# B&R Automation Studio project TD52 (part 80)

#### LamCtrPBC.h
```c
/********************************************************************
 * COPYRIGHT -- B&R Industrial Automation GmbH
 ********************************************************************
 * Program: LamCtrPBC
 * File: LamCtrPBC.h
 * Author: kafkama00
 * Last modified by: kafkama00
 * Created: Mon Oct 11 17:08:29 2021
 * Last modified: Wed Dec 01 09:46:51 2021
 * Model Version: 1.00
 * Description: Lambda controller for pressure based control engines
 * modified Comment: V0.01 11.10.2021 created for first tests
   V0.02 12.10.2021 added debug signals
   V0.03 17.11.2021 added distortion rejection
   V1.00 01.12.2021 remove distortion rejection, serial release DIA.NE V4.11
 ********************************************************************
 * Header for program LamCtrPBC
 ********************************************************************
 * Generated with B&R Automation Studio Target for Simulink V6.4.1
 * (ERT based)
 ********************************************************************/

#ifndef RTW_HEADER_LamCtrPBC_h_
#define RTW_HEADER_LamCtrPBC_h_
#include <math.h>
#include <string.h>
#ifndef LamCtrPBC_COMMON_INCLUDES_
# define LamCtrPBC_COMMON_INCLUDES_
#include "rtwtypes.h"
#include "zero_crossing_types.h"
#endif                                 /* LamCtrPBC_COMMON_INCLUDES_ */

#include "LamCtrPBC_types.h"
#include "lLamCtrPBC.h"
/* Beginning of Dynamic TypeDefs: */
/* End of Dynamic TypeDefs: */
#ifndef MIN
#define MIN(a,b)	((a) < (b) ? (a) : (b))
#endif

#ifndef MAX
#define MAX(a,b)	((a) > (b) ? (a) : (b))
#endif

#ifndef AST_ROUND
#define AST_ROUND(x) ((x)>=0?(long long)((x)+0.5):(long long)((x)-0.5))
#endif

#include "rt_defines.h"

/* Macros for accessing real-time model data structure */
#ifndef rtmGetBlockIO
# define rtmGetBlockIO(rtm)            ((rtm)->blockIO)
#endif

#ifndef rtmSetBlockIO
# define rtmSetBlockIO(rtm, val)       ((rtm)->blockIO = (val))
#endif

#ifndef rtmGetPrevZCSigState
# define rtmGetPrevZCSigState(rtm)     ((rtm)->prevZCSigState)
#endif

#ifndef rtmSetPrevZCSigState
# define rtmSetPrevZCSigState(rtm, val) ((rtm)->prevZCSigState = (val))
#endif

#ifndef rtmGetRootDWork
# define rtmGetRootDWork(rtm)          ((rtm)->dwork)
#endif

#ifndef rtmSetRootDWork
# define rtmSetRootDWork(rtm, val)     ((rtm)->dwork = (val))
#endif

#ifndef rtmGetU
# define rtmGetU(rtm)                  ((rtm)->inputs)
#endif

#ifndef rtmSetU
# define rtmSetU(rtm, val)             ((rtm)->inputs = (val))
#endif

#ifndef rtmGetY
# define rtmGetY(rtm)                  ((rtm)->outputs)
#endif

#ifndef rtmSetY
# define rtmSetY(rtm, val)             ((rtm)->outputs = (val))
#endif

#ifndef rtmGetErrorStatus
# define rtmGetErrorStatus(rtm)        ((rtm)->errorStatus)
#endif

#ifndef rtmSetErrorStatus
# define rtmSetErrorStatus(rtm, val)   ((rtm)->errorStatus = (val))
#endif

#ifndef MIN
#define MIN(a,b)                       ((a) < (b) ? (a) : (b))
#endif

#ifndef MAX
#define MAX(a,b)                       ((a) > (b) ? (a) : (b))
#endif

#ifndef AST_ROUND
#define AST_ROUND(x)                   ((x)>=0?(long long)((x)+0.5):(long long)((x)-0.5))
#endif

/* user code (top of header file) */
/***************************************************************************************************
 * COPYRIGHT -- INNIO Jenbacher GmbH & CO OG
 ****************************************************************************************************
 * Program:            LamCtrPBC
 * Author:             kafkama00
 * Created:            01.12.2021 09:46
 ****************************************************************************************************
 * MODEL INFORMATION
 ****************************************************************************************************
 * Model Name:         C:\Users\kafkama00\Documents\Git\LamCtrPBC\LamCtrPBC.slx
 * Model Version:      1.00
 * Simulink Version:   R2020a
 * B&R Target:         V6.4.1
 * Description:        Lambda controller for pressure based control engines
 ****************************************************************************************************
 * HISTORY
 ****************************************************************************************************
 * Last Modified By:   kafkama00
 * Last Modified Date: Wed Dec 01 09:46:42 2021
 * Modified Comment:   V0.01 11.10.2021 created for first tests
 *                     V0.02 12.10.2021 added debug signals
 *                     V0.03 17.11.2021 added distortion rejection
 *                     V1.00 01.12.2021 remove distortion rejection, serial release DIA.NE V4.11
 ****************************************************************************************************/

/* Block signals (default storage) */

/* Block states (default storage) for system '<Root>' */

/* Zero-crossing (trigger) state */

/* Invariant block signals (default storage) */

/* External inputs (root inport signals with default storage) */

/* External outputs (root outports fed by signals with default storage) */

/* Real-time Model Data Structure */

/* External data declarations for dependent source files */
extern const LamCtrPBC_IN_Bus LamCtrPBC_rtZLamCtrPBC_IN_Bus;/* LamCtrPBC_IN_Bus ground */
extern const LamCtrPBC_PARA_Bus LamCtrPBC_rtZLamCtrPBC_PARA_Bus;/* LamCtrPBC_PARA_Bus ground */
extern const LamCtrPBC_PERM_Bus LamCtrPBC_rtZLamCtrPBC_PERM_Bus;/* LamCtrPBC_PERM_Bus ground */
extern const LamCtrPBC_OUT_Bus LamCtrPBC_rtZLamCtrPBC_OUT_Bus;/* LamCtrPBC_OUT_Bus ground */
extern const LamCtrPBC_DBG_Bus LamCtrPBC_rtZLamCtrPBC_DBG_Bus;/* LamCtrPBC_DBG_Bus ground */
extern const ConstBlockIO_LamCtrPBC LamCtrPBC_ConstB;/* constant block i/o */

/* Model entry point functions */
extern void LamCtrPBC_initialize(RT_MODEL_LamCtrPBC *const LamCtrPBC_M, struct fLamCtrPBC* inst);
extern void LamCtrPBC_step(RT_MODEL_LamCtrPBC *const LamCtrPBC_M, struct fLamCtrPBC* inst);
extern void LamCtrPBC_terminate(RT_MODEL_LamCtrPBC *const LamCtrPBC_M, struct fLamCtrPBC* inst);

/*-
 * The generated code includes comments that allow you to trace directly
 * back to the appropriate location in the model.  The basic format
 * is <system>/block_name, where system is the system number (uniquely
 * assigned by Simulink) and block_name is the name of the block.
 *
 * Use the MATLAB hilite_system command to trace the generated code back
 * to the model.  For example,
 *
 * hilite_system('<S3>')    - opens system 3
 * hilite_system('<S3>/Kp') - opens and selects block Kp which resides in S3
 *
 * Here is the system hierarchy for this model
 *
 * '<Root>' : 'LamCtrPBC'
 * '<S1>'   : 'LamCtrPBC/Environment Controller'
 * '<S2>'   : 'LamCtrPBC/Environment Controller1'
 * '<S3>'   : 'LamCtrPBC/Environment Controller2'
 * '<S4>'   : 'LamCtrPBC/Filter2'
 * '<S5>'   : 'LamCtrPBC/Info'
 * '<S6>'   : 'LamCtrPBC/Saturation Dynamic'
 * '<S7>'   : 'LamCtrPBC/Filter2/Divisor'
 * '<S8>'   : 'LamCtrPBC/Filter2/Divisor/Data Type Conversion Inherited'
 */
#endif                                 /* RTW_HEADER_LamCtrPBC_h_ */
```

#### LamCtrPBC_data.c
```c
/********************************************************************
 * COPYRIGHT -- B&R Industrial Automation GmbH
 ********************************************************************
 * Program: LamCtrPBC
 * File: LamCtrPBC_data.c
 * Author: kafkama00
 * Last modified by: kafkama00
 * Created: Mon Oct 11 17:08:29 2021
 * Last modified: Wed Dec 01 09:46:51 2021
 * Model Version: 1.00
 * Description: Lambda controller for pressure based control engines
 * modified Comment: V0.01 11.10.2021 created for first tests
   V0.02 12.10.2021 added debug signals
   V0.03 17.11.2021 added distortion rejection
   V1.00 01.12.2021 remove distortion rejection, serial release DIA.NE V4.11
 ********************************************************************
 * Data for program LamCtrPBC
 ********************************************************************
 * Generated with B&R Automation Studio Target for Simulink V6.4.1
 * (ERT based)
 ********************************************************************/

#include "LamCtrPBC.h"
#include "LamCtrPBC_private.h"

/*  GLOBAL DATA DEFINITIONS */

/* Invariant block signals (default storage) */
const ConstBlockIO_LamCtrPBC LamCtrPBC_ConstB = {
  100U,                                /* '<S5>/Data Type Conversion3' */
  2.22044605E-16F                      /* '<S8>/Conversion' */
};
```

#### LamCtrPBC_private.h
```c
/********************************************************************
 * COPYRIGHT -- B&R Industrial Automation GmbH
 ********************************************************************
 * Program: LamCtrPBC
 * File: LamCtrPBC_private.h
 * Author: kafkama00
 * Last modified by: kafkama00
 * Created: Mon Oct 11 17:08:29 2021
 * Last modified: Wed Dec 01 09:46:51 2021
 * Model Version: 1.00
 * Description: Lambda controller for pressure based control engines
 * modified Comment: V0.01 11.10.2021 created for first tests
   V0.02 12.10.2021 added debug signals
   V0.03 17.11.2021 added distortion rejection
   V1.00 01.12.2021 remove distortion rejection, serial release DIA.NE V4.11
 ********************************************************************
 * Header for program LamCtrPBC
 ********************************************************************
 * Generated with B&R Automation Studio Target for Simulink V6.4.1
 * (ERT based)
 ********************************************************************/

#ifndef RTW_HEADER_LamCtrPBC_private_h_
#define RTW_HEADER_LamCtrPBC_private_h_
#include "rtwtypes.h"
#include "zero_crossing_types.h"
#include <bur/plctypes.h>
#ifndef MIN
#define MIN(a,b)                       ((a) < (b) ? (a) : (b))
#endif

#ifndef MAX
#define MAX(a,b)                       ((a) > (b) ? (a) : (b))
#endif

#ifndef AST_ROUND
#define AST_ROUND(x)                   ((x)>=0?(long long)((x)+0.5):(long long)((x)-0.5))
#endif
#endif                                 /* RTW_HEADER_LamCtrPBC_private_h_ */
```

#### LamCtrPBC_types.h
```c
/********************************************************************
 * COPYRIGHT -- B&R Industrial Automation GmbH
 ********************************************************************
 * Program: LamCtrPBC
 * File: LamCtrPBC_types.h
 * Author: kafkama00
 * Last modified by: kafkama00
 * Created: Mon Oct 11 17:08:29 2021
 * Last modified: Wed Dec 01 09:46:51 2021
 * Model Version: 1.00
 * Description: Lambda controller for pressure based control engines
 * modified Comment: V0.01 11.10.2021 created for first tests
   V0.02 12.10.2021 added debug signals
   V0.03 17.11.2021 added distortion rejection
   V1.00 01.12.2021 remove distortion rejection, serial release DIA.NE V4.11
 ********************************************************************
 * Header for program LamCtrPBC
 ********************************************************************
 * Generated with B&R Automation Studio Target for Simulink V6.4.1
 * (ERT based)
 ********************************************************************/

#ifndef RTW_HEADER_LamCtrPBC_types_h_
#define RTW_HEADER_LamCtrPBC_types_h_
#include "rtwtypes.h"

/* Model Code Variants */
#ifndef MIN
#define MIN(a,b)                       ((a) < (b) ? (a) : (b))
#endif

#ifndef MAX
#define MAX(a,b)                       ((a) > (b) ? (a) : (b))
#endif

#ifndef AST_ROUND
#define AST_ROUND(x)                   ((x)>=0?(long long)((x)+0.5):(long long)((x)-0.5))
#endif

/* Forward declaration for rtModel */

#endif                                 /* RTW_HEADER_LamCtrPBC_types_h_ */
```

#### fLamCtrPBC.c
```c
/********************************************************************
 * COPYRIGHT -- B&R Industrial Automation GmbH
 ********************************************************************
 * Program: LamCtrPBC
 * File: fLamCtrPBC.c
 * Author: kafkama00
 * Last modified by: kafkama00
 * Created: Mon Oct 11 17:08:29 2021
 * Last modified: Wed Dec 01 09:46:51 2021
 * Model Version: 1.00
 * Description: Lambda controller for pressure based control engines
 * modified Comment: V0.01 11.10.2021 created for first tests
   V0.02 12.10.2021 added debug signals
   V0.03 17.11.2021 added distortion rejection
   V1.00 01.12.2021 remove distortion rejection, serial release DIA.NE V4.11
 ********************************************************************
 * Implementation of program LamCtrPBC
 ********************************************************************
 * Generated with B&R Automation Studio Target for Simulink V6.4.1
 * (ERT based)
 ********************************************************************/

#include <bur/plctypes.h>
#include "LamCtrPBC.h"
#include "rtwtypes.h"

/* Defines */
#define SS_TERMINATE 4
#define SS_OUTPUT 3
#define SS_INITIALIZE 2

/*  Data Types */

/**************************** GLOBAL DATA *************************************/
/*  Definitions */

/*  Declarations  */

/***************************** FILE SCOPE DATA ********************************/

/*************************** FUNCTIONS ****************************************/
#ifdef __cplusplus

unsigned long bur_heap_size = 6553500;

#endif

/*LEGACYMODE_VARIABLES*/
void fLamCtrPBC(struct fLamCtrPBC* inst)
{
  tag_RTM_LamCtrPBC* const LamCtrPBC_M = &(inst)->bur_LamCtrPBC;
	inst->bur_LamCtrPBC.blockIO = &(inst)->bur_BlockIO_LamCtrPBC;
	inst->bur_LamCtrPBC.prevZCSigState = &(inst)->bur_PrevZCSigStates_LamCtrPBC;
	inst->bur_LamCtrPBC.inputs = &(inst)->bur_ExternalInputs_LamCtrPBC;
	inst->bur_LamCtrPBC.outputs = &(inst)->bur_ExternalOutputs_LamCtrPBC;
	inst->bur_LamCtrPBC.dwork = &(inst)->bur_D_Work_LamCtrPBC;

  switch (inst->ssMethodType)
  {
   case SS_INITIALIZE:
    /* call model initialize function */
    LamCtrPBC_initialize(LamCtrPBC_M, inst);
    break;

   case SS_OUTPUT:
    /* call model step function */
    LamCtrPBC_step(LamCtrPBC_M, inst);

    break;

   case SS_TERMINATE:
    /* call model terminate function */
    LamCtrPBC_terminate(LamCtrPBC_M, inst);
    break;
  }
}

/*****************************************************************************
   Function block sample time: 0.01s
 *****************************************************************************/

/*****************************************************************************
   B&R Automation Studio Target for Simulink Version: A6.4.1 (27-Apr-2021)
 *****************************************************************************/

/*======================== TOOL VERSION INFORMATION ==========================*
 * MATLAB 9.8 (R2020a)18-Nov-2019                                             *
 * Simulink 10.1 (R2020a)18-Nov-2019                                          *
 * Simulink Coder 9.3 (R2020a)18-Nov-2019                                     *
 * Embedded Coder 7.4 (R2020a)18-Nov-2019                                     *
 * Stateflow 10.2 (R2020a)18-Nov-2019                                         *
 *============================================================================*/

/*======================= LICENSE IN USE INFORMATION =========================*
 * matlab                                                                     *
 * matlab_coder                                                               *
 * real-time_workshop                                                         *
 * rtw_embedded_coder                                                         *
 * simulink                                                                   *
 *============================================================================*/
```

#### lLamCtrPBC.fun
```iecst
FUNCTION_BLOCK fLamCtrPBC
  VAR_INPUT
    ssMethodType: SINT;
  END_VAR
  VAR_INPUT
        In : LamCtrPBC_IN_Bus; (**)
  END_VAR
  VAR_INPUT
        Para : LamCtrPBC_PARA_Bus; (**)
  END_VAR
  VAR_INPUT
        Perm : LamCtrPBC_PERM_Bus; (**)
  END_VAR
  VAR_OUTPUT
        Out : LamCtrPBC_OUT_Bus; (**)
  END_VAR
  VAR_OUTPUT
        dbg : LamCtrPBC_DBG_Bus; (**)
  END_VAR
  VAR_OUTPUT
        Version : UDINT := 0; (**)
  END_VAR
	VAR
		bur_BlockIO_LamCtrPBC : BlockIO_LamCtrPBC;
	END_VAR
	VAR
		bur_PrevZCSigStates_LamCtrPBC : PrevZCSigStates_LamCtrPBC;
	END_VAR
	VAR
		bur_ExternalInputs_LamCtrPBC : ExternalInputs_LamCtrPBC;
	END_VAR
	VAR
		bur_ExternalOutputs_LamCtrPBC : ExternalOutputs_LamCtrPBC;
	END_VAR
	VAR
		bur_D_Work_LamCtrPBC : D_Work_LamCtrPBC;
	END_VAR
	VAR
		bur_LamCtrPBC : tag_RTM_LamCtrPBC;
	END_VAR
END_FUNCTION_BLOCK
```

#### lLamCtrPBC.typ
```iecst
TYPE
	LamCtrPBC_DBG_Bus :  STRUCT
		e_lam :  REAL; (*lambda deviation between set and estimation ()*)
		u :  REAL; (*lambda controller PBC offset output ()*)
		u_lim :  REAL; (*lambda controller PBC offset output limited  ()*)
		up_LamCtr :  REAL; (*proportional part of the lambda controller PBC output ()*)
		ui_LamCtr :  REAL; (*integral part of the lambda controller PBC output ()*)
		uAW_LamCtr :  REAL; (*anti windup of the lambda controller PBC ()*)
		u_PT1_smith :  REAL; (*signal after PT1 from smith predictor ()*)
		u_delay_smith :  REAL; (*signal after delay from smith predictor ()*)
		fb_smith :  REAL; (*feedback from smith predictor ()*)
	END_STRUCT;

	LamCtrPBC_IN_Bus :  STRUCT
		rLam_Set :  REAL; (*set lambda from high level controller (-)*)
		rLam_PBC :  REAL; (*lambda estimated from in-cylinder data (-)*)
		bReset :  BOOL; (*reset input of the lambda controller (-)*)
	END_STRUCT;

	LamCtrPBC_OUT_Bus :  STRUCT
		rLam_ref :  REAL; (*lambda reference for port injection opening duration calculation ()*)
	END_STRUCT;

	LamCtrPBC_PARA_Bus :  STRUCT
		rKp_LamCtr :  REAL; (*proportional gain for lambda controller PBC ()*)
		rKi_LamCtr :  REAL; (*integral gain for lambda controller PBC ()*)
		rKAW_LamCtr :  REAL; (*anti windup gain for lambda controller PBC ()*)
		rulim_LamCtr_up :  REAL; (*upper limit for lambda controller PBC output ()*)
		rulim_LamCtr_low :  REAL; (*lower limit for lambda controller PBC ()*)
	END_STRUCT;

	LamCtrPBC_PERM_Bus :  STRUCT
		iTd_smith_LamCtr :  SINT; (*delay time for smith predictor model ()*)
		rTi_smith_LamCtr :  REAL; (*filter time for smith predictor model ()*)
	END_STRUCT;

END_TYPE

TYPE
BlockIO_LamCtrPBC : STRUCT
	BusConversion_InsertedFor_BusOu : LamCtrPBC_DBG_Bus;
	BusInput1 : LamCtrPBC_PARA_Bus;
	BusInput : LamCtrPBC_IN_Bus;
	BusInput2 : LamCtrPBC_PERM_Bus;
	BusConversion_InsertedFor_Bus_b : LamCtrPBC_OUT_Bus;
	UnitDelay : UDINT;
END_STRUCT;
D_Work_LamCtrPBC : STRUCT
	Delay1_DSTATE : REAL;
	DiscreteTimeIntegrator_DSTATE : REAL;
	Delay_DSTATE : ARRAY[0..49] OF REAL;
	DiscreteTimeIntegrator_DSTATE_n : REAL;
	UnitDelay_DSTATE : UDINT;
	DiscreteTimeIntegrator_PrevRese : SINT;
	DiscreteTimeIntegrator_PrevRe_m : SINT;
	icLoad : USINT;
	icLoad_o : USINT;
	DiscreteTimeIntegrator_IC_LOADI : USINT;
END_STRUCT;
PrevZCSigStates_LamCtrPBC : STRUCT
	Delay1_Reset_ZCE : USINT;
END_STRUCT;
ConstBlockIO_LamCtrPBC : STRUCT
	DataTypeConversion3 : UDINT;
	Conversion : REAL;
END_STRUCT;
ExternalInputs_LamCtrPBC : STRUCT
	In : LamCtrPBC_IN_Bus;
	Para : LamCtrPBC_PARA_Bus;
	Perm : LamCtrPBC_PERM_Bus;
END_STRUCT;
ExternalOutputs_LamCtrPBC : STRUCT
	Out : LamCtrPBC_OUT_Bus;
	dbg : LamCtrPBC_DBG_Bus;
END_STRUCT;
tag_RTM_LamCtrPBC : STRUCT
	errorStatus : REFERENCE TO USINT;
	blockIO : REFERENCE TO BlockIO_LamCtrPBC;
	prevZCSigState : REFERENCE TO PrevZCSigStates_LamCtrPBC;
	inputs : REFERENCE TO ExternalInputs_LamCtrPBC;
	outputs : REFERENCE TO ExternalOutputs_LamCtrPBC;
	dwork : REFERENCE TO D_Work_LamCtrPBC;
END_STRUCT;
RT_MODEL_LamCtrPBC : tag_RTM_LamCtrPBC;

END_TYPE
TYPE
END_TYPE
```

#### lib_properties.txt
```
For manual assignment to hardware configuration please
add the following additional include directories:

\Logical\MATLAB_includes\R2020a\

And the following additional build options:

-lm -D MODEL=LamCtrPBC -D NUMST=1 -D NCSTATES=0 -D HAVESTDIO -D MODEL_HAS_DYNAMICALLY_LOADED_SFCNS=0 -D CLASSIC_INTERFACE=0 -D ALLOCATIONFCN=0 -D TID01EQ=0 -D TERMFCN=1 -D ONESTEPFCN=1 -D MAT_FILE=0 -D MULTI_INSTANCE_CODE=1 -D INTEGER_CODE=0 -D MT=0
```

#### rt_defines.h
```c
/********************************************************************
 * COPYRIGHT -- B&R Industrial Automation GmbH
 ********************************************************************
 * Program: LamCtrPBC
 * File: rt_defines.h
 * Author: kafkama00
 * Last modified by: kafkama00
 * Created: Mon Oct 11 17:08:29 2021
 * Last modified: Wed Dec 01 09:46:51 2021
 * Model Version: 1.00
 * Description: Lambda controller for pressure based control engines
 * modified Comment: V0.01 11.10.2021 created for first tests
   V0.02 12.10.2021 added debug signals
   V0.03 17.11.2021 added distortion rejection
   V1.00 01.12.2021 remove distortion rejection, serial release DIA.NE V4.11
 ********************************************************************
 * Header for program LamCtrPBC
 ********************************************************************
 * Generated with B&R Automation Studio Target for Simulink V6.4.1
 * (ERT based)
 ********************************************************************/

#ifndef RTW_HEADER_rt_defines_h_
#define RTW_HEADER_rt_defines_h_
#ifndef MIN
#define MIN(a,b)                       ((a) < (b) ? (a) : (b))
#endif

#ifndef MAX
#define MAX(a,b)                       ((a) > (b) ? (a) : (b))
#endif

#ifndef AST_ROUND
#define AST_ROUND(x)                   ((x)>=0?(long long)((x)+0.5):(long long)((x)-0.5))
#endif

/*===========*
 * Constants *
 *===========*/
#define RT_PI                          3.14159265358979323846
#define RT_PIF                         3.1415927F
#define RT_LN_10                       2.30258509299404568402
#define RT_LN_10F                      2.3025851F
#define RT_LOG10E                      0.43429448190325182765
#define RT_LOG10EF                     0.43429449F
#define RT_E                           2.7182818284590452354
#define RT_EF                          2.7182817F

/*
 * UNUSED_PARAMETER(x)
 *   Used to specify that a function parameter (argument) is required but not
 *   accessed by the function body.
 */
#ifndef UNUSED_PARAMETER
# if defined(__LCC__)
#   define UNUSED_PARAMETER(x)                                   /* do nothing */
# else

/*
 * This is the semi-ANSI standard way of indicating that an
 * unused function parameter is required.
 */
#   define UNUSED_PARAMETER(x)         (void) (x)
# endif
#endif
#endif                                 /* RTW_HEADER_rt_defines_h_ */
```

#### rtwtypes.h
```c
/********************************************************************
 * COPYRIGHT -- B&R Industrial Automation GmbH
 ********************************************************************
 * Program: LamCtrPBC
 * File: rtwtypes.h
 * Author: kafkama00
 * Last modified by: kafkama00
 * Created: Mon Oct 11 17:08:29 2021
 * Last modified: Wed Dec 01 09:46:51 2021
 * Model Version: 1.00
 * Description: Lambda controller for pressure based control engines
 * modified Comment: V0.01 11.10.2021 created for first tests
   V0.02 12.10.2021 added debug signals
   V0.03 17.11.2021 added distortion rejection
   V1.00 01.12.2021 remove distortion rejection, serial release DIA.NE V4.11
 ********************************************************************
 * Header for program LamCtrPBC
 ********************************************************************
 * Generated with B&R Automation Studio Target for Simulink V6.4.1
 * (ERT based)
 ********************************************************************/

#ifndef RTWTYPES_H
#define RTWTYPES_H

/* Logical type definitions */
#if (!defined(__cplusplus))
#  ifndef false
#   define false                       (0U)
#  endif

#  ifndef true
#   define true                        (1U)
#  endif
#endif

/*=======================================================================*
 * Target hardware information
 *   Device type: Intel->x86/Pentium
 *   Number of bits:     char:   8    short:   16    long:  32
 *                       long:  32
 *                       native word size:  32
 *   Byte ordering: LittleEndian
 *   Signed integer division rounds to: Zero
 *   Shift right on a signed integer as arithmetic shift: on
 *=======================================================================*/

/*=======================================================================*
 * Fixed width word size data types:                                     *
 *   int8_T, int16_T, int32_T     - signed 8, 16, or 32 bit integers     *
 *   uint8_T, uint16_T, uint32_T  - unsigned 8, 16, or 32 bit integers   *
 *   real32_T, real64_T           - 32 and 64 bit floating point numbers *
 *=======================================================================*/
typedef signed char int8_T;
typedef unsigned char uint8_T;
typedef short int16_T;
typedef unsigned short uint16_T;
typedef long int32_T;
typedef unsigned long uint32_T;
typedef float real32_T;
typedef double real64_T;

/*===========================================================================*
 * Generic type definitions: boolean_T, char_T, byte_T, int_T, uint_T,       *
 *                           real_T, time_T, ulong_T.                        *
 *===========================================================================*/
typedef double real_T;
typedef double time_T;
typedef unsigned char boolean_T;
typedef long int_T;
typedef unsigned long uint_T;
typedef unsigned long ulong_T;
typedef char char_T;
typedef unsigned char uchar_T;
typedef char_T byte_T;

/*=======================================================================*
 * Min and Max:                                                          *
 *   int8_T, int16_T, int32_T     - signed 8, 16, or 32 bit integers     *
 *   uint8_T, uint16_T, uint32_T  - unsigned 8, 16, or 32 bit integers   *
 *=======================================================================*/
#define MAX_int8_T                     ((int8_T)(127))
#define MIN_int8_T                     ((int8_T)(-128))
#define MAX_uint8_T                    ((uint8_T)(255U))
#define MAX_int16_T                    ((int16_T)(32767))
#define MIN_int16_T                    ((int16_T)(-32768))
#define MAX_uint16_T                   ((uint16_T)(65535U))
#define MAX_int32_T                    ((int32_T)(2147483647))
#define MIN_int32_T                    ((int32_T)(-2147483647-1))
#define MAX_uint32_T                   ((uint32_T)(0xFFFFFFFFU))

/* Block D-Work pointer type */
typedef void * pointer_T;

#endif                                 /* RTWTYPES_H */

#ifndef MIN
#define MIN(a,b)                       ((a) < (b) ? (a) : (b))
#endif

#ifndef MAX
#define MAX(a,b)                       ((a) > (b) ? (a) : (b))
#endif

#ifndef AST_ROUND
#define AST_ROUND(x)                   ((x)>=0?(long long)((x)+0.5):(long long)((x)-0.5))
#endif
```

#### zero_crossing_types.h
```c
/********************************************************************
 * COPYRIGHT -- B&R Industrial Automation GmbH
 ********************************************************************
 * Program: LamCtrPBC
 * File: zero_crossing_types.h
 * Author: kafkama00
 * Last modified by: kafkama00
 * Created: Mon Oct 11 17:08:29 2021
 * Last modified: Wed Dec 01 09:46:51 2021
 * Model Version: 1.00
 * Description: Lambda controller for pressure based control engines
 * modified Comment: V0.01 11.10.2021 created for first tests
   V0.02 12.10.2021 added debug signals
   V0.03 17.11.2021 added distortion rejection
   V1.00 01.12.2021 remove distortion rejection, serial release DIA.NE V4.11
 ********************************************************************
 * Header for program LamCtrPBC
 ********************************************************************
 * Generated with B&R Automation Studio Target for Simulink V6.4.1
 * (ERT based)
 ********************************************************************/

#ifndef ZERO_CROSSING_TYPES_H
#define ZERO_CROSSING_TYPES_H
#include "rtwtypes.h"

/* Trigger directions: falling, either, and rising */
typedef enum {
  FALLING_ZERO_CROSSING = -1,
  ANY_ZERO_CROSSING = 0,
  RISING_ZERO_CROSSING = 1
} ZCDirection;

/* Previous state of a trigger signal */
typedef uint8_T ZCSigState;

/* Initial value of a trigger zero crossing signal */
#define UNINITIALIZED_ZCSIG            0x03U
#define NEG_ZCSIG                      0x02U
#define POS_ZCSIG                      0x01U
#define ZERO_ZCSIG                     0x00U

/* Current state of a trigger signal */
typedef enum {
  FALLING_ZCEVENT = -1,
  NO_ZCEVENT = 0,
  RISING_ZCEVENT = 1
} ZCEventType;

#endif                                 /* ZERO_CROSSING_TYPES_H */

#ifndef MIN
#define MIN(a,b)                       ((a) < (b) ? (a) : (b))
#endif

#ifndef MAX
#define MAX(a,b)                       ((a) > (b) ? (a) : (b))
#endif

#ifndef AST_ROUND
#define AST_ROUND(x)                   ((x)>=0?(long long)((x)+0.5):(long long)((x)-0.5))
#endif
```

### Library Logical/EngineController/Lib_EC/lTrStRed (ANSIC, version 1.00.0)

#### TrStRed.c
```c
/********************************************************************
 * COPYRIGHT -- B&R Industrial Automation GmbH
 ********************************************************************
 * Program: TrStRed
 * File: TrStRed.c
 * Author: 105055527
 * Last modified by: maranen00
 * Created: Mon Sep 05 18:14:57 2016
 * Last modified: Mon Dec 06 12:59:10 2021
 * Model Version: 0.3.0
 * Description: Thermal reactor start time reduction function

   Outstandings:
   -------------
   - NA
 * modified Comment: V0.1.0 18.05.2021 Maran   TrStRed function first draft
   V0.1.1 27.05.2021 Maran   added limitation based on cyl. EG max temp. above setpoint
   V0.1.2 02.08.2021 Maran   added half load factor for function limit range
   V0.2.0 15.11.2021 Maran   added saturation limits to control error for the closed loop integrator (PERM parameters)
   V0.3.0 06.12.2021 Maran   removed unused logic in controller block; added filtered value of monitoring variables in debug interface
 ********************************************************************
 * Implementation of program TrStRed
 ********************************************************************
 * Generated with B&R Automation Studio Target for Simulink V6.3.1
 * (ERT based)
 ********************************************************************/

#include "TrStRed.h"
#include "TrStRed_private.h"

/*  Defines */

/*  Data Types */

/**************************** GLOBAL DATA *************************************/
/*  Definitions */

/*  Declarations  */

/***************************** FILE SCOPE DATA ********************************/

/*************************** FUNCTIONS ****************************************/

/* Lookup Binary Search Utility BINARYSEARCH_real32_T */
void BINARYSEARCH_real32_T(uint32_T *piLeft, uint32_T *piRght, real32_T u, const
  real32_T *pData, uint32_T iHi, struct fTrStRed* inst)
{
  /* Find the location of current input value in the data table. */
  *piLeft = 0U;
  *piRght = iHi;
  if (u <= pData[0] ) {
    /* Less than or equal to the smallest point in the table. */
    *piRght = 0U;
  } else if (u >= pData[iHi] ) {
    /* Greater than or equal to the largest point in the table. */
    *piLeft = iHi;
  } else {
    uint32_T i;

    /* Do a binary search. */
    while (( *piRght - *piLeft ) > 1U ) {
      /* Get the average of the left and right indices using to Floor rounding. */
      i = (*piLeft + *piRght) >> 1;

      /* Move either the right index or the left index so that */
      /*  LeftDataPoint <= CurrentValue < RightDataPoint */
      if (u < pData[i] ) {
        *piRght = i;
      } else {
        *piLeft = i;
      }
    }
  }
}

/* Lookup Utility LookUp_real32_T_real32_T */
void LookUp_real32_T_real32_T(real32_T *pY, const real32_T *pYData, real32_T u,
  const real32_T *pUData, uint32_T iHi, struct fTrStRed* inst)
{
  uint32_T iLeft;
  uint32_T iRght;
  BINARYSEARCH_real32_T( &(iLeft), &(iRght), u, pUData, iHi, inst);

  {
    real32_T lambda;
    if (pUData[iRght] > pUData[iLeft] ) {
      real32_T num;
      real32_T den;
      den = pUData[iRght];
      den -= pUData[iLeft];
      num = u;
      num -= pUData[iLeft];
      lambda = num / den;
    } else {
      lambda = 0.0F;
    }

    {
      real32_T yLeftCast;
      real32_T yRghtCast;
      yLeftCast = pYData[iLeft];
      yRghtCast = pYData[iRght];
      yLeftCast += lambda * ( yRghtCast - yLeftCast );
      (*pY) = yLeftCast;
    }
  }
}

/*
 * System initialize for atomic system:
 *    '<S6>/Filter'
 *    '<S6>/Filter1'
 */
void TrStRed_Filter_Init(rtDW_Filter_TrStRed *localDW, struct fTrStRed* inst)
{
  /* InitializeConditions for DiscreteIntegrator: '<S17>/Discrete-Time Integrator' */
  localDW->DiscreteTimeIntegrator_IC_LOADI = 1U;
}

/*
 * Output and update for atomic system:
 *    '<S6>/Filter'
 *    '<S6>/Filter1'
 */
void TrStRed_Filter(real32_T rtu_in, real32_T rtu_T_filt, boolean_T rtu_reset,
                    rtB_Filter_TrStRed *localB, rtDW_Filter_TrStRed *localDW, struct fTrStRed* inst)
{
  boolean_T rtb_RelationalOperator_bj;
  boolean_T rtb_LogicalOperator_f;
  real32_T tmp;

  /* RelationalOperator: '<S17>/Relational Operator' incorporates:
   *  Constant: '<S17>/Constant'
   */
  rtb_RelationalOperator_bj = (rtu_T_filt > 0.0F);

  /* Logic: '<S17>/Logical Operator' incorporates:
   *  Logic: '<S17>/Logical Operator1'
   */
  rtb_LogicalOperator_f = (rtu_reset || (!rtb_RelationalOperator_bj));

  /* DiscreteIntegrator: '<S17>/Discrete-Time Integrator' */
  if (localDW->DiscreteTimeIntegrator_IC_LOADI != 0) {
    localDW->DiscreteTimeIntegrator_DSTATE = rtu_in;
  }

  if (rtb_LogicalOperator_f || (localDW->DiscreteTimeIntegrator_PrevRese != 0))
  {
    localDW->DiscreteTimeIntegrator_DSTATE = rtu_in;
  }

  /* Switch: '<S17>/Switch' incorporates:
   *  DiscreteIntegrator: '<S17>/Discrete-Time Integrator'
   */
  if (rtb_RelationalOperator_bj) {
    localB->Switch = localDW->DiscreteTimeIntegrator_DSTATE;
  } else {
    localB->Switch = rtu_in;
  }

  /* End of Switch: '<S17>/Switch' */

  /* Update for DiscreteIntegrator: '<S17>/Discrete-Time Integrator' */
  localDW->DiscreteTimeIntegrator_IC_LOADI = 0U;

  /* Switch: '<S28>/Switch' incorporates:
   *  Abs: '<S28>/Abs'
   *  RelationalOperator: '<S28>/Relational Operator'
   */
  if (2.22044605E-16F >= (real32_T)fabs(rtu_T_filt)) {
    tmp = 2.22044605E-16F;
  } else {
    tmp = rtu_T_filt;
  }

  /* End of Switch: '<S28>/Switch' */

  /* Update for DiscreteIntegrator: '<S17>/Discrete-Time Integrator' incorporates:
   *  Product: '<S17>/Divide4'
   *  Sum: '<S17>/Sum4'
   */
  localDW->DiscreteTimeIntegrator_DSTATE += (rtu_in -
    localDW->DiscreteTimeIntegrator_DSTATE) / tmp * 0.01F;
  localDW->DiscreteTimeIntegrator_PrevRese = (int8_T)rtb_LogicalOperator_f;
}

/*
 * Output and update for atomic system:
 *    '<S8>/TON'
 *    '<S10>/TON'
 */
void TrStRed_TON(boolean_T rtu_IN, uint16_T rtu_PT, rtB_TON_TrStRed *localB,
                 rtDW_TON_TrStRed *localDW, struct fTrStRed* inst)
{
  boolean_T rtb_LogicalOperator2;
  boolean_T rtb_RelationalOperator_a;
  uint32_T tmp;

  /* Logic: '<S34>/Logical Operator2' */
  rtb_LogicalOperator2 = !rtu_IN;

  /* DiscreteIntegrator: '<S34>/Discrete-Time Integrator' */
  if (rtb_LogicalOperator2 || (localDW->DiscreteTimeIntegrator_PrevRese != 0)) {
    localDW->DiscreteTimeIntegrator_DSTATE = 0U;
  }

  /* RelationalOperator: '<S34>/Relational Operator' incorporates:
   *  DiscreteIntegrator: '<S34>/Discrete-Time Integrator'
   */
  tmp = localDW->DiscreteTimeIntegrator_DSTATE * 41943U;
  rtb_RelationalOperator_a = (((tmp & 32U) != 0U) + (tmp >> 6) >= ((uint32_T)
    rtu_PT << 16));

  /* Logic: '<S34>/Logical Operator3' */
  localB->LogicalOperator3 = (rtb_RelationalOperator_a && rtu_IN);

  /* Update for DiscreteIntegrator: '<S34>/Discrete-Time Integrator' incorporates:
   *  Logic: '<S34>/Logical Operator'
   *  Logic: '<S34>/Logical Operator1'
   */
  localDW->DiscreteTimeIntegrator_DSTATE = (uint16_T)((uint32_T)
    ((!rtb_RelationalOperator_a) && rtu_IN) +
    localDW->DiscreteTimeIntegrator_DSTATE);
  localDW->DiscreteTimeIntegrator_PrevRese = (int8_T)rtb_LogicalOperator2;
}

/* Model step function */
void TrStRed_step(RT_MODEL_TrStRed *const TrStRed_M, struct fTrStRed* inst)
{
  struct BlockIO_TrStRed *TrStRed_B = ((struct BlockIO_TrStRed *) TrStRed_M->blockIO);
  struct D_Work_TrStRed *TrStRed_DWork = ((struct D_Work_TrStRed *) TrStRed_M->dwork);
  struct PrevZCSigStates_TrStRed *TrStRed_PrevZCSigState = ((struct PrevZCSigStates_TrStRed *)
    TrStRed_M->prevZCSigState);
  ExternalOutputs_TrStRed *TrStRed_Y = (ExternalOutputs_TrStRed *)
    TrStRed_M->outputs;
  int32_T rowIdx;
  real32_T rtb_Switch2;
  real32_T rtb_Switch2_e;
  real32_T rtb_Subtract5;
  real32_T rtb_Product;
  real32_T rtb_Saturation1;
  real32_T rtb_Product1;
  boolean_T rtb_RelationalOperator_c;
  boolean_T rtb_LowerRelop1_c;
  real32_T rtb_DiscreteTimeIntegrator;
  real32_T rtb_Subtract;
  real32_T rtb_TmpSignalConversionAtLookup[2];
  real32_T rtb_TmpSignalConversionAtLook_f[2];
  boolean_T rtb_Logic_b_idx_0;
  boolean_T rtb_Logic_idx_0;
  boolean_T rtb_Logic_e_idx_0;
  real32_T u0;
  real32_T u0_0;
  real32_T u0_1;
  real32_T u0_2;
  uint32_T rtb_Logic_idx_0_tmp;
  boolean_T rtb_Logic_idx_0_tmp_0;

  /* S-Function (bur_bus_in): '<Root>/Bus Input1' */
  TrStRed_B->BusInput1 = inst->Perm;

  /* Product: '<S20>/delta rise limit' incorporates:
   *  SampleTimeMath: '<S20>/sample time'
   *  Switch: '<S4>/Environment Switch'
   *
   * About '<S20>/sample time':
   *  y = K where K = ( w * Ts )
   */
  rtb_Switch2 = TrStRed_B->BusInput1.rCA_RateLimit * 0.01F;

  /* S-Function (bur_bus_in): '<Root>/Bus Input2' */
  TrStRed_B->BusInput2 = inst->In;

  /* Switch: '<S2>/Environment Switch' */
  rtb_Product1 = TrStRed_B->BusInput2.rP_Set_Norm;

  /* Outputs for Atomic SubSystem: '<S8>/TON' */
  /* Logic: '<S8>/Logical Operator' incorporates:
   *  Abs: '<S8>/Abs'
   *  RelationalOperator: '<S8>/Relational Operator'
   *  Sum: '<S8>/Sum'
   *  Switch: '<S2>/Environment Switch'
   *  Switch: '<S4>/Environment Switch'
   */
  TrStRed_TON(TrStRed_B->BusInput2.bTrStRed_active && ((real32_T)fabs
    (TrStRed_B->BusInput2.rP_Norm - rtb_Product1) <=
    TrStRed_B->BusInput1.rP_diffThres_Steady),
              TrStRed_B->BusInput1.iTimerDelay_Steady, &TrStRed_B->TON,
              &TrStRed_DWork->TON, inst);

  /* End of Outputs for SubSystem: '<S8>/TON' */

  /* CombinatorialLogic: '<S37>/Logic' incorporates:
   *  CombinatorialLogic: '<S36>/Logic'
   *  Logic: '<S9>/Logical Operator2'
   *  Switch: '<S2>/Environment Switch'
   */
  rtb_Logic_idx_0_tmp = (uint32_T)(TrStRed_B->BusInput2.bTrStRed_active &&
    TrStRed_B->TON.LogicalOperator3) << 1;

  /* Logic: '<S9>/NOT1' incorporates:
   *  Logic: '<S6>/Logical Operator'
   *  Switch: '<S2>/Environment Switch'
   */
  rtb_Logic_idx_0_tmp_0 = !TrStRed_B->BusInput2.bTrStRed_active;

  /* CombinatorialLogic: '<S37>/Logic' incorporates:
   *  Logic: '<S9>/NOT1'
   *  Memory: '<S37>/Memory'
   */
  rtb_Logic_idx_0 = TrStRed_ConstP.pooled10[((rtb_Logic_idx_0_tmp +
    rtb_Logic_idx_0_tmp_0) << 1) + TrStRed_DWork->Memory_PreviousInput];

  /* CombinatorialLogic: '<S36>/Logic' incorporates:
   *  Memory: '<S36>/Memory'
   *  Switch: '<S2>/Environment Switch'
   */
  rowIdx = (int32_T)(((rtb_Logic_idx_0_tmp + TrStRed_B->BusInput2.bCycleReset) <<
                      1) + TrStRed_DWork->Memory_PreviousInput_o);
  rtb_Logic_b_idx_0 = TrStRed_ConstP.pooled10[(uint32_T)rowIdx];

  /* Outputs for Atomic SubSystem: '<S10>/TON' */
  /* Switch: '<S2>/Environment Switch' incorporates:
   *  Switch: '<S4>/Environment Switch'
   */
  TrStRed_TON(TrStRed_B->BusInput2.bThR_RelGas, TrStRed_B->BusInput1.iStopTimer,
              &TrStRed_B->TON_k, &TrStRed_DWork->TON_k, inst);

  /* End of Outputs for SubSystem: '<S10>/TON' */

  /* CombinatorialLogic: '<S38>/Logic' incorporates:
   *  CombinatorialLogic: '<S36>/Logic'
   *  Logic: '<S10>/Logical Operator'
   *  Memory: '<S38>/Memory'
   *  Switch: '<S2>/Environment Switch'
   */
  rowIdx = (int32_T)(((((uint32_T)(TrStRed_ConstP.pooled10[(uint32_T)rowIdx] &&
    TrStRed_B->TON_k.LogicalOperator3) << 1) + TrStRed_B->BusInput2.bCycleReset)
                      << 1) + TrStRed_DWork->Memory_PreviousInput_l);
  rtb_Logic_e_idx_0 = TrStRed_ConstP.pooled10[(uint32_T)rowIdx];

  /* Logic: '<Root>/NOT8' incorporates:
   *  CombinatorialLogic: '<S38>/Logic'
   *  Logic: '<Root>/NOT1'
   */
  rtb_LowerRelop1_c = ((!rtb_Logic_idx_0) || TrStRed_ConstP.pooled10[(uint32_T)
                       rowIdx]);

  /* Logic: '<Root>/NOT6' incorporates:
   *  Logic: '<Root>/Logical Operator1'
   *  Logic: '<Root>/NOT7'
   *  Switch: '<S2>/Environment Switch'
   *  UnitDelay: '<Root>/Unit Delay'
   */
  rtb_RelationalOperator_c = ((TrStRed_DWork->UnitDelay_DSTATE_j &&
    rtb_LowerRelop1_c) || TrStRed_B->BusInput2.bReset || (!rtb_Logic_b_idx_0));

  /* DiscreteIntegrator: '<S1>/Discrete-Time Integrator' incorporates:
   *  Switch: '<S2>/Environment Switch'
   */
  if (TrStRed_DWork->DiscreteTimeIntegrator_IC_LOADI != 0) {
    TrStRed_DWork->ITCtrUi = TrStRed_B->BusInput2.rCA_Ign_UpLim;
  }

  if (rtb_RelationalOperator_c ||
      (TrStRed_DWork->DiscreteTimeIntegrator_PrevRese != 0)) {
    TrStRed_DWork->ITCtrUi = TrStRed_B->BusInput2.rCA_Ign_UpLim;
  }

  rtb_DiscreteTimeIntegrator = TrStRed_DWork->ITCtrUi;

  /* Product: '<S21>/delta rise limit' incorporates:
   *  Gain: '<S6>/Gain1'
   *  SampleTimeMath: '<S21>/sample time'
   *  Switch: '<S4>/Environment Switch'
   *
   * About '<S21>/sample time':
   *  y = K where K = ( w * Ts )
   */
  rtb_Switch2_e = 100.0F * TrStRed_B->BusInput1.rCA_RateLimit * 0.01F;

  /* Gain: '<S6>/misfire_Lim [%]' incorporates:
   *  Switch: '<S4>/Environment Switch'
   */
  rtb_Product = 100.0F * TrStRed_B->BusInput1.rMisfire_Lim;

  /* Sum: '<S6>/Subtract5' incorporates:
   *  Gain: '<S6>/misfire [%]'
   *  Switch: '<S2>/Environment Switch'
   */
  rtb_Subtract5 = rtb_Product - 100.0F * TrStRed_B->BusInput2.rMisfire_level;

  /* Switch: '<S13>/Switch' incorporates:
   *  Abs: '<S13>/Abs'
   *  RelationalOperator: '<S13>/Relational Operator'
   */
  if (0.1F >= (real32_T)fabs(rtb_Product)) {
    rtb_Product = 0.1F;
  }

  /* End of Switch: '<S13>/Switch' */

  /* Product: '<S6>/Divide3' */
  rtb_Product = rtb_Subtract5 / rtb_Product;

  /* Saturate: '<S6>/Saturation3' */
  if (rtb_Product > 1.0F) {
    rtb_Product = 1.0F;
  } else {
    if (rtb_Product < 0.0F) {
      rtb_Product = 0.0F;
    }
  }

  /* End of Saturate: '<S6>/Saturation3' */

  /* Outputs for Atomic SubSystem: '<S6>/Filter1' */
  /* Switch: '<S2>/Environment Switch' incorporates:
   *  Switch: '<S4>/Environment Switch'
   */
  TrStRed_Filter(TrStRed_B->BusInput2.rIgnVolt_Max,
                 TrStRed_B->BusInput1.rFiltConst_IgnVolt, rtb_Logic_idx_0_tmp_0,
                 &TrStRed_B->Filter1, &TrStRed_DWork->Filter1, inst);

  /* End of Outputs for SubSystem: '<S6>/Filter1' */

  /* S-Function (bur_bus_in): '<Root>/Bus Input' */
  TrStRed_B->BusInput = inst->Para;

  /* Outputs for Atomic SubSystem: '<S6>/Filter' */
  /* Switch: '<S2>/Environment Switch' incorporates:
   *  Switch: '<S4>/Environment Switch'
   */
  TrStRed_Filter(TrStRed_B->BusInput2.rPr_Leanox_Dev,
                 TrStRed_B->BusInput1.rFiltConst_LxDev, rtb_Logic_idx_0_tmp_0,
                 &TrStRed_B->Filter, &TrStRed_DWork->Filter, inst);

  /* End of Outputs for SubSystem: '<S6>/Filter' */

  /* Gain: '<S6>/Gain' incorporates:
   *  Switch: '<S4>/Environment Switch'
   */
  rtb_Saturation1 = 0.5F * TrStRed_B->BusInput1.rPr_LxDev_Lim;

  /* Switch: '<S14>/Switch' incorporates:
   *  Abs: '<S14>/Abs'
   *  RelationalOperator: '<S14>/Relational Operator'
   */
  if (0.1F >= (real32_T)fabs(rtb_Saturation1)) {
    rtb_Saturation1 = 0.1F;
  }

  /* End of Switch: '<S14>/Switch' */

  /* Product: '<S6>/Divide4' incorporates:
   *  Sum: '<S6>/Subtract6'
   *  Switch: '<S4>/Environment Switch'
   */
  u0 = (TrStRed_B->BusInput1.rPr_LxDev_Lim - TrStRed_B->Filter.Switch) /
    rtb_Saturation1;

  /* Sum: '<S6>/Subtract4' incorporates:
   *  Switch: '<S2>/Environment Switch'
   *  Switch: '<S4>/Environment Switch'
   */
  rtb_Saturation1 = TrStRed_B->BusInput2.rT_EG_MaxLimit -
    TrStRed_B->BusInput1.rT_EG_Max_LimOffset;

  /* Sum: '<S6>/Subtract1' incorporates:
   *  Switch: '<S2>/Environment Switch'
   */
  rtb_Subtract5 = rtb_Saturation1 - TrStRed_B->BusInput2.rT_EG_CylMax;

  /* MinMax: '<S6>/Max' */
  if (rtb_Subtract5 <= 0.0F) {
    rtb_Subtract5 = 0.0F;
  }

  /* End of MinMax: '<S6>/Max' */

  /* Sum: '<Root>/Subtract' incorporates:
   *  Switch: '<S2>/Environment Switch'
   *  Switch: '<S3>/Environment Switch'
   */
  rtb_Subtract = TrStRed_B->BusInput2.rT_EG_MaxLimit -
    TrStRed_B->BusInput.rT_EG_Max_LimMarg;

  /* Sum: '<S6>/Subtract3' */
  rtb_Saturation1 -= rtb_Subtract;

  /* MinMax: '<S6>/Max1' */
  if (rtb_Saturation1 <= 0.0F) {
    rtb_Saturation1 = 0.0F;
  }

  /* End of MinMax: '<S6>/Max1' */

  /* Switch: '<S12>/Switch' incorporates:
   *  Abs: '<S12>/Abs'
   *  RelationalOperator: '<S12>/Relational Operator'
   */
  if (0.1F >= rtb_Saturation1) {
    rtb_Saturation1 = 0.1F;
  }

  /* End of Switch: '<S12>/Switch' */

  /* Product: '<S6>/Divide1' */
  rtb_Saturation1 = rtb_Subtract5 / rtb_Saturation1;

  /* Saturate: '<S6>/Saturation1' */
  if (rtb_Saturation1 > 1.0F) {
    rtb_Saturation1 = 1.0F;
  }

  /* End of Saturate: '<S6>/Saturation1' */

  /* Abs: '<S16>/Abs' incorporates:
   *  Switch: '<S4>/Environment Switch'
   */
  rtb_Subtract5 = (real32_T)fabs(TrStRed_B->BusInput1.rT_EGbTC_LimMarg);

  /* Switch: '<S16>/Switch' incorporates:
   *  RelationalOperator: '<S16>/Relational Operator'
   *  Switch: '<S4>/Environment Switch'
   */
  if (0.1F >= rtb_Subtract5) {
    rtb_Subtract5 = 0.1F;
  } else {
    rtb_Subtract5 = TrStRed_B->BusInput1.rT_EGbTC_LimMarg;
  }

  /* End of Switch: '<S16>/Switch' */

  /* Switch: '<S11>/Switch' incorporates:
   *  Abs: '<S11>/Abs'
   *  RelationalOperator: '<S11>/Relational Operator'
   *  Switch: '<S4>/Environment Switch'
   */
  if (0.1F >= (real32_T)fabs(TrStRed_B->BusInput1.rIgnVolt_LimMarg)) {
    u0_1 = 0.1F;
  } else {
    u0_1 = TrStRed_B->BusInput1.rIgnVolt_LimMarg;
  }

  /* End of Switch: '<S11>/Switch' */

  /* Product: '<S6>/Divide' incorporates:
   *  Sum: '<S6>/Subtract2'
   *  Sum: '<S6>/Sum'
   *  Switch: '<S3>/Environment Switch'
   *  Switch: '<S4>/Environment Switch'
   */
  u0_0 = ((TrStRed_B->BusInput.rIgnVoltMax_Lim +
           TrStRed_B->BusInput1.rIgnVolt_LimMarg) - TrStRed_B->Filter1.Switch) /
    u0_1;

  /* Switch: '<S15>/Switch' incorporates:
   *  Abs: '<S15>/Abs'
   *  RelationalOperator: '<S15>/Relational Operator'
   *  Switch: '<S4>/Environment Switch'
   */
  if (0.1F >= (real32_T)fabs(TrStRed_B->BusInput1.rT_EG_Avg_LimMarg)) {
    u0_1 = 0.1F;
  } else {
    u0_1 = TrStRed_B->BusInput1.rT_EG_Avg_LimMarg;
  }

  /* End of Switch: '<S15>/Switch' */

  /* Product: '<S6>/Divide5' incorporates:
   *  Sum: '<S6>/Subtract7'
   *  Switch: '<S2>/Environment Switch'
   *  Switch: '<S3>/Environment Switch'
   */
  u0_1 = (TrStRed_B->BusInput.rT_EG_Avg_HiLim -
          TrStRed_B->BusInput2.rT_EG_CylAvg) / u0_1;

  /* Product: '<S6>/Divide6' incorporates:
   *  Sum: '<S6>/Subtract8'
   *  Switch: '<S2>/Environment Switch'
   *  Switch: '<S3>/Environment Switch'
   */
  u0_2 = (TrStRed_B->BusInput.rT_EGbTC_HiLim - TrStRed_B->BusInput2.rT_EGbTC) /
    rtb_Subtract5;

  /* Saturate: '<S6>/Saturation' */
  if (u0_0 > 1.0F) {
    u0_0 = 1.0F;
  } else {
    if (u0_0 < 0.0F) {
      u0_0 = 0.0F;
    }
  }

  /* End of Saturate: '<S6>/Saturation' */

  /* Saturate: '<S6>/Saturation6' */
  if (u0 > 1.0F) {
    u0 = 1.0F;
  } else {
    if (u0 < 0.0F) {
      u0 = 0.0F;
    }
  }

  /* End of Saturate: '<S6>/Saturation6' */

  /* Saturate: '<S6>/Saturation8' */
  if (u0_1 > 1.0F) {
    u0_1 = 1.0F;
  } else {
    if (u0_1 < 0.0F) {
      u0_1 = 0.0F;
    }
  }

  /* End of Saturate: '<S6>/Saturation8' */

  /* Saturate: '<S6>/Saturation10' */
  if (u0_2 > 1.0F) {
    u0_2 = 1.0F;
  } else {
    if (u0_2 < 0.0F) {
      u0_2 = 0.0F;
    }
  }

  /* End of Saturate: '<S6>/Saturation10' */

  /* Product: '<S6>/Product' */
  rtb_Product = rtb_Product * u0_0 * u0 * u0_1 * rtb_Saturation1 * u0_2;

  /* Product: '<S6>/Product2' incorporates:
   *  Switch: '<S3>/Environment Switch'
   */
  rtb_Product *= TrStRed_B->BusInput.rCA_TrStRed_LowLimit;

  /* Delay: '<S21>/Delay' */
  if ((((TrStRed_PrevZCSigState->Delay_Reset_ZCE == 1) != (int32_T)
        rtb_RelationalOperator_c) && (TrStRed_PrevZCSigState->Delay_Reset_ZCE !=
        3)) || rtb_RelationalOperator_c) {
    TrStRed_DWork->icLoad = 1U;
  }

  TrStRed_PrevZCSigState->Delay_Reset_ZCE = rtb_RelationalOperator_c;
  if (TrStRed_DWork->icLoad != 0) {
    TrStRed_DWork->Delay_DSTATE = rtb_Product;
  }

  /* Sum: '<S21>/Difference Inputs1' incorporates:
   *  Delay: '<S21>/Delay'
   *  Switch: '<S21>/etaVolConst'
   */
  rtb_Product -= TrStRed_DWork->Delay_DSTATE;

  /* Switch: '<S33>/Switch2' incorporates:
   *  RelationalOperator: '<S33>/LowerRelop1'
   */
  if (rtb_Product <= rtb_Switch2_e) {
    /* Product: '<S21>/delta fall limit' incorporates:
     *  Product: '<S6>/Product3'
     *  SampleTimeMath: '<S21>/sample time'
     *  Switch: '<S4>/Environment Switch'
     *  UnaryMinus: '<S6>/Unary Minus1'
     *
     * About '<S21>/sample time':
     *  y = K where K = ( w * Ts )
     */
    rtb_Switch2_e = -(TrStRed_B->BusInput1.rCA_RateLimit *
                      TrStRed_B->BusInput1.rLimitsReleaseFactor) * 0.01F;

    /* Switch: '<S33>/Switch' incorporates:
     *  RelationalOperator: '<S33>/UpperRelop'
     */
    if (rtb_Product >= rtb_Switch2_e) {
      rtb_Switch2_e = rtb_Product;
    }

    /* End of Switch: '<S33>/Switch' */
  }

  /* End of Switch: '<S33>/Switch2' */

  /* Sum: '<S21>/Difference Inputs2' incorporates:
   *  Delay: '<S21>/Delay'
   */
  rtb_Switch2_e += TrStRed_DWork->Delay_DSTATE;

  /* SignalConversion generated from: '<S6>/Lookup Table Dynamic' incorporates:
   *  Constant: '<S6>/Constant2'
   *  Constant: '<S6>/Constant3'
   */
  rtb_TmpSignalConversionAtLookup[0] = 0.5F;
  rtb_TmpSignalConversionAtLookup[1] = 0.9F;

  /* SignalConversion generated from: '<S6>/Lookup Table Dynamic' incorporates:
   *  Constant: '<S6>/Constant4'
   *  Switch: '<S3>/Environment Switch'
   */
  rtb_TmpSignalConversionAtLook_f[0] =
    TrStRed_B->BusInput.rGain_TrStRed_halfLoadLim;
  rtb_TmpSignalConversionAtLook_f[1] = 1.0F;

  /* S-Function (sfix_look1_dyn): '<S6>/Lookup Table Dynamic' */
  /* Dynamic Look-Up Table Block: '<S6>/Lookup Table Dynamic'
   * Input0  Data Type:  Floating Point real32_T
   * Input1  Data Type:  Floating Point real32_T
   * Input2  Data Type:  Floating Point real32_T
   * Output0 Data Type:  Floating Point real32_T
   * Lookup Method: Linear_Endpoint
   *
   */
  LookUp_real32_T_real32_T( &(rtb_Subtract5), &rtb_TmpSignalConversionAtLook_f[0],
    rtb_Product1, &rtb_TmpSignalConversionAtLookup[0], 1U, inst);

  /* Product: '<S6>/Product1' */
  rtb_Product1 = rtb_Switch2_e * rtb_Subtract5;

  /* Switch: '<S19>/Switch2' incorporates:
   *  DiscreteIntegrator: '<S1>/Discrete-Time Integrator'
   *  RelationalOperator: '<S19>/LowerRelop1'
   *  RelationalOperator: '<S19>/UpperRelop'
   *  Switch: '<S19>/Switch'
   *  Switch: '<S2>/Environment Switch'
   */
  if (TrStRed_DWork->ITCtrUi > TrStRed_B->BusInput2.rCA_Ign_UpLim) {
    rtb_Subtract5 = TrStRed_B->BusInput2.rCA_Ign_UpLim;
  } else if (TrStRed_DWork->ITCtrUi < rtb_Product1) {
    /* Switch: '<S19>/Switch' */
    rtb_Subtract5 = rtb_Product1;
  } else {
    rtb_Subtract5 = TrStRed_DWork->ITCtrUi;
  }

  /* End of Switch: '<S19>/Switch2' */

  /* Switch: '<S6>/Switch1' incorporates:
   *  Switch: '<S2>/Environment Switch'
   */
  if (rtb_LowerRelop1_c) {
    rtb_Product = TrStRed_B->BusInput2.rCA_Ign_UpLim;
  } else {
    rtb_Product = rtb_Subtract5;
  }

  /* End of Switch: '<S6>/Switch1' */

  /* Delay: '<S20>/Delay' */
  if ((((TrStRed_PrevZCSigState->Delay_Reset_ZCE_l == 1) != (int32_T)
        rtb_RelationalOperator_c) && (TrStRed_PrevZCSigState->Delay_Reset_ZCE_l
        != 3)) || rtb_RelationalOperator_c) {
    TrStRed_DWork->icLoad_l = 1U;
  }

  TrStRed_PrevZCSigState->Delay_Reset_ZCE_l = rtb_RelationalOperator_c;
  if (TrStRed_DWork->icLoad_l != 0) {
    TrStRed_DWork->Delay_DSTATE_b = rtb_Product;
  }

  /* Sum: '<S20>/Difference Inputs1' incorporates:
   *  Delay: '<S20>/Delay'
   *  Switch: '<S20>/etaVolConst'
   */
  rtb_Product -= TrStRed_DWork->Delay_DSTATE_b;

  /* Switch: '<S32>/Switch2' incorporates:
   *  RelationalOperator: '<S32>/LowerRelop1'
   */
  if (rtb_Product <= rtb_Switch2) {
    /* Product: '<S20>/delta fall limit' incorporates:
     *  SampleTimeMath: '<S20>/sample time'
     *  Switch: '<S4>/Environment Switch'
     *  UnaryMinus: '<S6>/Unary Minus'
     *
     * About '<S20>/sample time':
     *  y = K where K = ( w * Ts )
     */
    rtb_Switch2 = -TrStRed_B->BusInput1.rCA_RateLimit * 0.01F;

    /* Switch: '<S32>/Switch' incorporates:
     *  RelationalOperator: '<S32>/UpperRelop'
     */
    if (rtb_Product >= rtb_Switch2) {
      rtb_Switch2 = rtb_Product;
    }

    /* End of Switch: '<S32>/Switch' */
  }

  /* End of Switch: '<S32>/Switch2' */

  /* Sum: '<S20>/Difference Inputs2' incorporates:
   *  Delay: '<S20>/Delay'
   */
  rtb_Switch2 += TrStRed_DWork->Delay_DSTATE_b;

  /* BusCreator: '<Root>/Bus Creator1' incorporates:
   *  CombinatorialLogic: '<S38>/Logic'
   *  Outport: '<Root>/Out'
   */
  TrStRed_Y->Out.rCA_IP_Lim = rtb_Switch2;
  TrStRed_Y->Out.bCycleStarted = rtb_Logic_b_idx_0;
  TrStRed_Y->Out.bCycleCompleted = TrStRed_ConstP.pooled10[(uint32_T)rowIdx];
  TrStRed_Y->Out.bTrStRed_Stop = rtb_RelationalOperator_c;

  /* Sum: '<Root>/Subtract1' incorporates:
   *  Switch: '<S2>/Environment Switch'
   */
  rtb_Subtract -= TrStRed_B->BusInput2.rT_EG_CylMax;

  /* Switch: '<S7>/Switch2' incorporates:
   *  RelationalOperator: '<S7>/LowerRelop1'
   *  RelationalOperator: '<S7>/UpperRelop'
   *  Switch: '<S4>/Environment Switch'
   *  Switch: '<S7>/Switch'
   */
  if (rtb_Subtract > TrStRed_B->BusInput1.rT_CtrlError_UpLim) {
    rtb_Subtract = TrStRed_B->BusInput1.rT_CtrlError_UpLim;
  } else {
    if (rtb_Subtract < TrStRed_B->BusInput1.rT_CtrlError_LowLim) {
      /* Switch: '<S7>/Switch' */
      rtb_Subtract = TrStRed_B->BusInput1.rT_CtrlError_LowLim;
    }
  }

  /* End of Switch: '<S7>/Switch2' */

  /* BusCreator: '<Root>/Bus Creator4' incorporates:
   *  DiscreteIntegrator: '<S1>/Discrete-Time Integrator'
   *  Outport: '<Root>/dbg'
   *  RelationalOperator: '<S6>/Relational Operator'
   */
  TrStRed_Y->dbg.bInternalLimitAct = (TrStRed_DWork->ITCtrUi != rtb_Subtract5);

  /* UnitDelay: '<S1>/Unit Delay1' */
  rtb_Subtract5 = TrStRed_DWork->UnitDelay1_DSTATE;

  /* Sum: '<S1>/Subtract1' incorporates:
   *  Switch: '<S2>/Environment Switch'
   */
  rtb_Subtract5 = TrStRed_B->BusInput2.rCA_IgnP_relAw - rtb_Subtract5;

  /* Product: '<S1>/Product3' incorporates:
   *  Switch: '<S4>/Environment Switch'
   */
  rtb_Subtract5 *= TrStRed_B->BusInput1.rCtrl_kAw;

  /* Sum: '<S1>/Sum' incorporates:
   *  Gain: '<Root>/Gain'
   */
  rtb_Subtract5 += -rtb_Subtract;

  /* Product: '<S1>/Product1' incorporates:
   *  Switch: '<S4>/Environment Switch'
   */
  rtb_Product = TrStRed_B->BusInput1.rCtrl_ki * rtb_Subtract5;

  /* BusCreator: '<Root>/Bus Creator4' incorporates:
   *  DiscreteIntegrator: '<S1>/Discrete-Time Integrator'
   *  Outport: '<Root>/dbg'
   */
  TrStRed_Y->dbg.rT_CtrlError = rtb_Subtract;
  TrStRed_Y->dbg.rCA_IP_Lim_preSat = TrStRed_DWork->ITCtrUi;
  TrStRed_Y->dbg.rCtrl_Int_InputPreGain = rtb_Subtract5;
  TrStRed_Y->dbg.rPr_Leanox_Dev_filt = TrStRed_B->Filter.Switch;
  TrStRed_Y->dbg.rIgnVolt_Max_filt = TrStRed_B->Filter1.Switch;
  TrStRed_Y->dbg.rCtrl_IntegrInput = rtb_Product;
  TrStRed_Y->dbg.bSteadyState = TrStRed_B->TON.LogicalOperator3;
  TrStRed_Y->dbg.rCA_LowLimit_Act = rtb_Product1;

  /* S-Function (bur_bus_out): '<Root>/Bus Output' incorporates:
   *  Outport: '<Root>/Out'
   */
  inst->Out = TrStRed_Y->Out;

  /* S-Function (bur_bus_out): '<Root>/Bus Output1' incorporates:
   *  Outport: '<Root>/dbg'
   */
  inst->Dbg = TrStRed_Y->dbg;

  /* Bias: '<Root>/Bias' incorporates:
   *  Switch: '<S2>/Environment Switch'
   */
  rtb_Subtract5 = TrStRed_B->BusInput2.rCA_Ign_UpLim + -0.01F;

  /* UnitDelay: '<S5>/Unit Delay' */
  TrStRed_B->UnitDelay = TrStRed_DWork->UnitDelay_DSTATE;

  /* S-Function (bur_out): '<Root>/Output1' */
  inst->Version = TrStRed_B->UnitDelay;

  /* Update for Memory: '<S37>/Memory' */
  TrStRed_DWork->Memory_PreviousInput = rtb_Logic_idx_0;

  /* Update for Memory: '<S36>/Memory' */
  TrStRed_DWork->Memory_PreviousInput_o = rtb_Logic_b_idx_0;

  /* Update for Memory: '<S38>/Memory' */
  TrStRed_DWork->Memory_PreviousInput_l = rtb_Logic_e_idx_0;

  /* Update for UnitDelay: '<Root>/Unit Delay' incorporates:
   *  RelationalOperator: '<Root>/Relational Operator'
   */
  TrStRed_DWork->UnitDelay_DSTATE_j = (rtb_Switch2 >= rtb_Subtract5);

  /* Update for DiscreteIntegrator: '<S1>/Discrete-Time Integrator' */
  TrStRed_DWork->DiscreteTimeIntegrator_IC_LOADI = 0U;
  TrStRed_DWork->ITCtrUi += 0.01F * rtb_Product;
  TrStRed_DWork->DiscreteTimeIntegrator_PrevRese = (int8_T)
    rtb_RelationalOperator_c;

  /* Update for Delay: '<S21>/Delay' */
  TrStRed_DWork->icLoad = 0U;
  TrStRed_DWork->Delay_DSTATE = rtb_Switch2_e;

  /* Update for Delay: '<S20>/Delay' */
  TrStRed_DWork->icLoad_l = 0U;
  TrStRed_DWork->Delay_DSTATE_b = rtb_Switch2;

  /* Update for UnitDelay: '<S1>/Unit Delay1' */
  TrStRed_DWork->UnitDelay1_DSTATE = rtb_DiscreteTimeIntegrator;

  /* Update for UnitDelay: '<S5>/Unit Delay' */
  TrStRed_DWork->UnitDelay_DSTATE = 30U;
}

/* Model initialize function */
void TrStRed_initialize(RT_MODEL_TrStRed *const TrStRed_M, struct fTrStRed* inst)
{
  struct D_Work_TrStRed *TrStRed_DWork = ((struct D_Work_TrStRed *) TrStRed_M->dwork);
  struct PrevZCSigStates_TrStRed *TrStRed_PrevZCSigState = ((struct PrevZCSigStates_TrStRed *)
    TrStRed_M->prevZCSigState);
  TrStRed_PrevZCSigState->Delay_Reset_ZCE = UNINITIALIZED_ZCSIG;
  TrStRed_PrevZCSigState->Delay_Reset_ZCE_l = UNINITIALIZED_ZCSIG;

  /* InitializeConditions for DiscreteIntegrator: '<S1>/Discrete-Time Integrator' */
  TrStRed_DWork->DiscreteTimeIntegrator_IC_LOADI = 1U;

  /* InitializeConditions for Delay: '<S21>/Delay' */
  TrStRed_DWork->icLoad = 1U;

  /* InitializeConditions for Delay: '<S20>/Delay' */
  TrStRed_DWork->icLoad_l = 1U;

  /* SystemInitialize for Atomic SubSystem: '<S6>/Filter1' */
  TrStRed_Filter_Init(&TrStRed_DWork->Filter1, inst);

  /* End of SystemInitialize for SubSystem: '<S6>/Filter1' */

  /* SystemInitialize for Atomic SubSystem: '<S6>/Filter' */
  TrStRed_Filter_Init(&TrStRed_DWork->Filter, inst);

  /* End of SystemInitialize for SubSystem: '<S6>/Filter' */
}

/* Model terminate function */
void TrStRed_terminate(RT_MODEL_TrStRed *const TrStRed_M, struct fTrStRed* inst)
{
  /* (no terminate code required) */
  UNUSED_PARAMETER(TrStRed_M);
}

/*======================== TOOL VERSION INFORMATION ==========================*
 * MATLAB 9.8 (R2020a)18-Nov-2019                                             *
 * Simulink 10.1 (R2020a)18-Nov-2019                                          *
 * Simulink Coder 9.3 (R2020a)18-Nov-2019                                     *
 * Embedded Coder 7.4 (R2020a)18-Nov-2019                                     *
 * Stateflow 10.2 (R2020a)18-Nov-2019                                         *
 *============================================================================*/

/*======================= LICENSE IN USE INFORMATION =========================*
 * matlab                                                                     *
 * matlab_coder                                                               *
 * real-time_workshop                                                         *
 * rtw_embedded_coder                                                         *
 * simulink                                                                   *
 *============================================================================*/
```

#### TrStRed.h
```c
/********************************************************************
 * COPYRIGHT -- B&R Industrial Automation GmbH
 ********************************************************************
 * Program: TrStRed
 * File: TrStRed.h
 * Author: 105055527
 * Last modified by: maranen00
 * Created: Mon Sep 05 18:14:57 2016
 * Last modified: Mon Dec 06 12:59:10 2021
 * Model Version: 0.3.0
 * Description: Thermal reactor start time reduction function

   Outstandings:
   -------------
   - NA
 * modified Comment: V0.1.0 18.05.2021 Maran   TrStRed function first draft
   V0.1.1 27.05.2021 Maran   added limitation based on cyl. EG max temp. above setpoint
   V0.1.2 02.08.2021 Maran   added half load factor for function limit range
   V0.2.0 15.11.2021 Maran   added saturation limits to control error for the closed loop integrator (PERM parameters)
   V0.3.0 06.12.2021 Maran   removed unused logic in controller block; added filtered value of monitoring variables in debug interface
 ********************************************************************
 * Header for program TrStRed
 ********************************************************************
 * Generated with B&R Automation Studio Target for Simulink V6.3.1
 * (ERT based)
 ********************************************************************/

#ifndef RTW_HEADER_TrStRed_h_
#define RTW_HEADER_TrStRed_h_
#include <math.h>
#ifndef TrStRed_COMMON_INCLUDES_
# define TrStRed_COMMON_INCLUDES_
#include "rtwtypes.h"
#include "zero_crossing_types.h"
#endif                                 /* TrStRed_COMMON_INCLUDES_ */

#include "TrStRed_types.h"
#include "lTrStRed.h"
/* Beginning of Dynamic TypeDefs: */
/* End of Dynamic TypeDefs: */
#ifndef MIN
#define MIN(a,b)	((a) < (b) ? (a) : (b))
#endif

#ifndef MAX
#define MAX(a,b)	((a) > (b) ? (a) : (b))
#endif

#ifndef AST_ROUND
#define AST_ROUND(x) ((x)>=0?(long long)((x)+0.5):(long long)((x)-0.5))
#endif

#include "rt_defines.h"

/* Macros for accessing real-time model data structure */
#ifndef rtmGetBlockIO
# define rtmGetBlockIO(rtm)            ((rtm)->blockIO)
#endif

#ifndef rtmSetBlockIO
# define rtmSetBlockIO(rtm, val)       ((rtm)->blockIO = (val))
#endif

#ifndef rtmGetPrevZCSigState
# define rtmGetPrevZCSigState(rtm)     ((rtm)->prevZCSigState)
#endif

#ifndef rtmSetPrevZCSigState
# define rtmSetPrevZCSigState(rtm, val) ((rtm)->prevZCSigState = (val))
#endif

#ifndef rtmGetRootDWork
# define rtmGetRootDWork(rtm)          ((rtm)->dwork)
#endif

#ifndef rtmSetRootDWork
# define rtmSetRootDWork(rtm, val)     ((rtm)->dwork = (val))
#endif

#ifndef rtmGetU
# define rtmGetU(rtm)                  ((rtm)->inputs)
#endif

#ifndef rtmSetU
# define rtmSetU(rtm, val)             ((rtm)->inputs = (val))
#endif

#ifndef rtmGetY
# define rtmGetY(rtm)                  ((rtm)->outputs)
#endif

#ifndef rtmSetY
# define rtmSetY(rtm, val)             ((rtm)->outputs = (val))
#endif

#ifndef rtmGetErrorStatus
# define rtmGetErrorStatus(rtm)        ((rtm)->errorStatus)
#endif

#ifndef rtmSetErrorStatus
# define rtmSetErrorStatus(rtm, val)   ((rtm)->errorStatus = (val))
#endif

#ifndef MIN
#define MIN(a,b)                       ((a) < (b) ? (a) : (b))
#endif

#ifndef MAX
#define MAX(a,b)                       ((a) > (b) ? (a) : (b))
#endif

#ifndef AST_ROUND
#define AST_ROUND(x)                   ((x)>=0?(long long)((x)+0.5):(long long)((x)-0.5))
#endif

/* user code (top of header file) */
/***************************************************************************************************
 * COPYRIGHT -- INNIO Jenbacher GmbH & CO OG
 ****************************************************************************************************
 * Program:            TrStRed
 * Author:             maranen00
 * Created:            06.12.2021 12:59
 ****************************************************************************************************
 * MODEL INFORMATION
 ****************************************************************************************************
 * Model Name:         C:\Git\Cl-Air_start_time_reduction\02_Modeling_and_Auto-code_generation\TrStRed.slx
 * Model Version:      0.3.0
 * Simulink Version:   R2020a
 * B&R Target:         V6.3.1
 * Description:        Thermal reactor start time reduction function
 *
 *                     Outstandings:
 *                     -------------
 *                     - NA
 ****************************************************************************************************
 * HISTORY
 ****************************************************************************************************
 * Last Modified By:   maranen00
 * Last Modified Date: Mon Dec 06 12:55:28 2021
 * Modified Comment:   V0.1.0 18.05.2021 Maran   TrStRed function first draft
 *                     V0.1.1 27.05.2021 Maran   added limitation based on cyl. EG max temp. above setpoint
 *                     V0.1.2 02.08.2021 Maran   added half load factor for function limit range
 *                     V0.2.0 15.11.2021 Maran   added saturation limits to control error for the closed loop integrator (PERM parameters)
 *                     V0.3.0 06.12.2021 Maran   removed unused logic in controller block; added filtered value of monitoring variables in debug interface
 ****************************************************************************************************/

/* Block signals for system '<S6>/Filter' */

/* Block states (default storage) for system '<S6>/Filter' */

/* Block signals for system '<S8>/TON' */

/* Block states (default storage) for system '<S8>/TON' */

/* Block signals (default storage) */

/* Block states (default storage) for system '<Root>' */

/* Zero-crossing (trigger) state */

/* Invariant block signals for system '<S6>/Filter' */

/* Invariant block signals (default storage) */

/* Constant parameters (default storage) */

/* External inputs (root inport signals with default storage) */

/* External outputs (root outports fed by signals with default storage) */

/* Real-time Model Data Structure */

extern const ConstBlockIO_TrStRed TrStRed_ConstB;/* constant block i/o */

/* Constant parameters (default storage) */
extern const ConstParam_TrStRed TrStRed_ConstP;

/* Model entry point functions */
extern void TrStRed_initialize(RT_MODEL_TrStRed *const TrStRed_M, struct fTrStRed* inst);
extern void TrStRed_step(RT_MODEL_TrStRed *const TrStRed_M, struct fTrStRed* inst);
extern void TrStRed_terminate(RT_MODEL_TrStRed *const TrStRed_M, struct fTrStRed* inst);

/*-
 * The generated code includes comments that allow you to trace directly
 * back to the appropriate location in the model.  The basic format
 * is <system>/block_name, where system is the system number (uniquely
 * assigned by Simulink) and block_name is the name of the block.
 *
 * Use the MATLAB hilite_system command to trace the generated code back
 * to the model.  For example,
 *
 * hilite_system('<S3>')    - opens system 3
 * hilite_system('<S3>/Kp') - opens and selects block Kp which resides in S3
 *
 * Here is the system hierarchy for this model
 *
 * '<Root>' : 'TrStRed'
 * '<S1>'   : 'TrStRed/Ctrl'
 * '<S2>'   : 'TrStRed/Environment Controller'
 * '<S3>'   : 'TrStRed/Environment Controller1'
 * '<S4>'   : 'TrStRed/Environment Controller2'
 * '<S5>'   : 'TrStRed/Info'
 * '<S6>'   : 'TrStRed/Limitation'
 * '<S7>'   : 'TrStRed/Saturation Dynamic'
 * '<S8>'   : 'TrStRed/SteadyState'
 * '<S9>'   : 'TrStRed/TrStRed_started'
 * '<S10>'  : 'TrStRed/TrStRed_stopping'
 * '<S11>'  : 'TrStRed/Limitation/Divisor'
 * '<S12>'  : 'TrStRed/Limitation/Divisor1'
 * '<S13>'  : 'TrStRed/Limitation/Divisor3'
 * '<S14>'  : 'TrStRed/Limitation/Divisor4'
 * '<S15>'  : 'TrStRed/Limitation/Divisor5'
 * '<S16>'  : 'TrStRed/Limitation/Divisor6'
 * '<S17>'  : 'TrStRed/Limitation/Filter'
 * '<S18>'  : 'TrStRed/Limitation/Filter1'
 * '<S19>'  : 'TrStRed/Limitation/Saturation Dynamic'
 * '<S20>'  : 'TrStRed/Limitation/rateLimit'
 * '<S21>'  : 'TrStRed/Limitation/rateLimit1'
 * '<S22>'  : 'TrStRed/Limitation/Divisor/Data Type Conversion Inherited'
 * '<S23>'  : 'TrStRed/Limitation/Divisor1/Data Type Conversion Inherited'
 * '<S24>'  : 'TrStRed/Limitation/Divisor3/Data Type Conversion Inherited'
 * '<S25>'  : 'TrStRed/Limitation/Divisor4/Data Type Conversion Inherited'
 * '<S26>'  : 'TrStRed/Limitation/Divisor5/Data Type Conversion Inherited'
 * '<S27>'  : 'TrStRed/Limitation/Divisor6/Data Type Conversion Inherited'
 * '<S28>'  : 'TrStRed/Limitation/Filter/Divisor'
 * '<S29>'  : 'TrStRed/Limitation/Filter/Divisor/Data Type Conversion Inherited'
 * '<S30>'  : 'TrStRed/Limitation/Filter1/Divisor'
 * '<S31>'  : 'TrStRed/Limitation/Filter1/Divisor/Data Type Conversion Inherited'
 * '<S32>'  : 'TrStRed/Limitation/rateLimit/Saturation Dynamic'
 * '<S33>'  : 'TrStRed/Limitation/rateLimit1/Saturation Dynamic'
 * '<S34>'  : 'TrStRed/SteadyState/TON'
 * '<S35>'  : 'TrStRed/SteadyState/TON/Data Type Conversion Inherited'
 * '<S36>'  : 'TrStRed/TrStRed_started/S-R Flip-Flop'
 * '<S37>'  : 'TrStRed/TrStRed_started/S-R Flip-Flop1'
 * '<S38>'  : 'TrStRed/TrStRed_stopping/S-R Flip-Flop'
 * '<S39>'  : 'TrStRed/TrStRed_stopping/TON'
 * '<S40>'  : 'TrStRed/TrStRed_stopping/TON/Data Type Conversion Inherited'
 */
#endif                                 /* RTW_HEADER_TrStRed_h_ */
```

#### TrStRed_data.c
```c
/********************************************************************
 * COPYRIGHT -- B&R Industrial Automation GmbH
 ********************************************************************
 * Program: TrStRed
 * File: TrStRed_data.c
 * Author: 105055527
 * Last modified by: maranen00
 * Created: Mon Sep 05 18:14:57 2016
 * Last modified: Mon Dec 06 12:59:10 2021
 * Model Version: 0.3.0
 * Description: Thermal reactor start time reduction function

   Outstandings:
   -------------
   - NA
 * modified Comment: V0.1.0 18.05.2021 Maran   TrStRed function first draft
   V0.1.1 27.05.2021 Maran   added limitation based on cyl. EG max temp. above setpoint
   V0.1.2 02.08.2021 Maran   added half load factor for function limit range
   V0.2.0 15.11.2021 Maran   added saturation limits to control error for the closed loop integrator (PERM parameters)
   V0.3.0 06.12.2021 Maran   removed unused logic in controller block; added filtered value of monitoring variables in debug interface
 ********************************************************************
 * Data for program TrStRed
 ********************************************************************
 * Generated with B&R Automation Studio Target for Simulink V6.3.1
 * (ERT based)
 ********************************************************************/

#include "TrStRed.h"
#include "TrStRed_private.h"

/*  GLOBAL DATA DEFINITIONS */

/* Invariant block signals (default storage) */
const ConstBlockIO_TrStRed TrStRed_ConstB = {
  /* Start of '<S6>/Filter1' */
  {
    2.22044605E-16F                    /* '<S31>/Conversion' */
  }
  ,

  /* End of '<S6>/Filter1' */

  /* Start of '<S6>/Filter' */
  {
    2.22044605E-16F                    /* '<S29>/Conversion' */
  }
  /* End of '<S6>/Filter' */
};

/* Constant parameters (default storage) */
const ConstParam_TrStRed TrStRed_ConstP = {
  /* Pooled Parameter (Expression: [0 1;1 0;0 1;0 1;1 0;1 0;0 0;0 0])
   * Referenced by:
   *   '<S36>/Logic'
   *   '<S37>/Logic'
   *   '<S38>/Logic'
   */
  { 0, 1, 0, 0, 1, 1, 0, 0, 1, 0, 1, 1, 0, 0, 0, 0 }
};
```

#### TrStRed_private.h
```c
/********************************************************************
 * COPYRIGHT -- B&R Industrial Automation GmbH
 ********************************************************************
 * Program: TrStRed
 * File: TrStRed_private.h
 * Author: 105055527
 * Last modified by: maranen00
 * Created: Mon Sep 05 18:14:57 2016
 * Last modified: Mon Dec 06 12:59:10 2021
 * Model Version: 0.3.0
 * Description: Thermal reactor start time reduction function

   Outstandings:
   -------------
   - NA
 * modified Comment: V0.1.0 18.05.2021 Maran   TrStRed function first draft
   V0.1.1 27.05.2021 Maran   added limitation based on cyl. EG max temp. above setpoint
   V0.1.2 02.08.2021 Maran   added half load factor for function limit range
   V0.2.0 15.11.2021 Maran   added saturation limits to control error for the closed loop integrator (PERM parameters)
   V0.3.0 06.12.2021 Maran   removed unused logic in controller block; added filtered value of monitoring variables in debug interface
 ********************************************************************
 * Header for program TrStRed
 ********************************************************************
 * Generated with B&R Automation Studio Target for Simulink V6.3.1
 * (ERT based)
 ********************************************************************/

#ifndef RTW_HEADER_TrStRed_private_h_
#define RTW_HEADER_TrStRed_private_h_
#include "rtwtypes.h"
#include "zero_crossing_types.h"
#include "TrStRed.h"
#include <bur/plctypes.h>
#ifndef UCHAR_MAX
#include <limits.h>
#endif

#if ( UCHAR_MAX != (0xFFU) ) || ( SCHAR_MAX != (0x7F) )
#error Code was generated for compiler with different sized uchar/char. \
Consider adjusting Test hardware word size settings on the \
Hardware Implementation pane to match your compiler word sizes as \
defined in limits.h of the compiler. Alternatively, you can \
select the Test hardware is the same as production hardware option and \
select the Enable portable word sizes option on the Code Generation > \
Verification pane for ERT based targets, which will disable the \
preprocessor word size checks.
#endif

#if ( USHRT_MAX != (0xFFFFU) ) || ( SHRT_MAX != (0x7FFF) )
#error Code was generated for compiler with different sized ushort/short. \
Consider adjusting Test hardware word size settings on the \
Hardware Implementation pane to match your compiler word sizes as \
defined in limits.h of the compiler. Alternatively, you can \
select the Test hardware is the same as production hardware option and \
select the Enable portable word sizes option on the Code Generation > \
Verification pane for ERT based targets, which will disable the \
preprocessor word size checks.
#endif

#if ( UINT_MAX != (0xFFFFFFFFU) ) || ( INT_MAX != (0x7FFFFFFF) )
#error Code was generated for compiler with different sized uint/int. \
Consider adjusting Test hardware word size settings on the \
Hardware Implementation pane to match your compiler word sizes as \
defined in limits.h of the compiler. Alternatively, you can \
select the Test hardware is the same as production hardware option and \
select the Enable portable word sizes option on the Code Generation > \
Verification pane for ERT based targets, which will disable the \
preprocessor word size checks.
#endif

#if ( ULONG_MAX != (0xFFFFFFFFU) ) || ( LONG_MAX != (0x7FFFFFFF) )
#error Code was generated for compiler with different sized ulong/long. \
Consider adjusting Test hardware word size settings on the \
Hardware Implementation pane to match your compiler word sizes as \
defined in limits.h of the compiler. Alternatively, you can \
select the Test hardware is the same as production hardware option and \
select the Enable portable word sizes option on the Code Generation > \
Verification pane for ERT based targets, which will disable the \
preprocessor word size checks.
#endif

#ifndef MIN
#define MIN(a,b)                       ((a) < (b) ? (a) : (b))
#endif

#ifndef MAX
#define MAX(a,b)                       ((a) > (b) ? (a) : (b))
#endif

#ifndef AST_ROUND
#define AST_ROUND(x)                   ((x)>=0?(long long)((x)+0.5):(long long)((x)-0.5))
#endif

void BINARYSEARCH_real32_T(uint32_T *piLeft, uint32_T *piRght, real32_T u, const
  real32_T *pData, uint32_T iHi, struct fTrStRed* inst);
void LookUp_real32_T_real32_T(real32_T *pY, const real32_T *pYData, real32_T u,
  const real32_T *pUData, uint32_T iHi, struct fTrStRed* inst);
extern void TrStRed_Filter_Init(rtDW_Filter_TrStRed *localDW, struct fTrStRed* inst);
extern void TrStRed_Filter(real32_T rtu_in, real32_T rtu_T_filt, boolean_T
  rtu_reset, rtB_Filter_TrStRed *localB, rtDW_Filter_TrStRed *localDW, struct fTrStRed* inst);
extern void TrStRed_TON(boolean_T rtu_IN, uint16_T rtu_PT, rtB_TON_TrStRed
  *localB, rtDW_TON_TrStRed *localDW, struct fTrStRed* inst);

#endif                                 /* RTW_HEADER_TrStRed_private_h_ */
```

#### TrStRed_types.h
```c
/********************************************************************
 * COPYRIGHT -- B&R Industrial Automation GmbH
 ********************************************************************
 * Program: TrStRed
 * File: TrStRed_types.h
 * Author: 105055527
 * Last modified by: maranen00
 * Created: Mon Sep 05 18:14:57 2016
 * Last modified: Mon Dec 06 12:59:10 2021
 * Model Version: 0.3.0
 * Description: Thermal reactor start time reduction function

   Outstandings:
   -------------
   - NA
 * modified Comment: V0.1.0 18.05.2021 Maran   TrStRed function first draft
   V0.1.1 27.05.2021 Maran   added limitation based on cyl. EG max temp. above setpoint
   V0.1.2 02.08.2021 Maran   added half load factor for function limit range
   V0.2.0 15.11.2021 Maran   added saturation limits to control error for the closed loop integrator (PERM parameters)
   V0.3.0 06.12.2021 Maran   removed unused logic in controller block; added filtered value of monitoring variables in debug interface
 ********************************************************************
 * Header for program TrStRed
 ********************************************************************
 * Generated with B&R Automation Studio Target for Simulink V6.3.1
 * (ERT based)
 ********************************************************************/

#ifndef RTW_HEADER_TrStRed_types_h_
#define RTW_HEADER_TrStRed_types_h_
#include "rtwtypes.h"

/* Model Code Variants */
#ifndef MIN
#define MIN(a,b)                       ((a) < (b) ? (a) : (b))
#endif

#ifndef MAX
#define MAX(a,b)                       ((a) > (b) ? (a) : (b))
#endif

#ifndef AST_ROUND
#define AST_ROUND(x)                   ((x)>=0?(long long)((x)+0.5):(long long)((x)-0.5))
#endif

/* Forward declaration for rtModel */

#endif                                 /* RTW_HEADER_TrStRed_types_h_ */
```

#### fTrStRed.c
```c
/********************************************************************
 * COPYRIGHT -- B&R Industrial Automation GmbH
 ********************************************************************
 * Program: TrStRed
 * File: fTrStRed.c
 * Author: 105055527
 * Last modified by: maranen00
 * Created: Mon Sep 05 18:14:57 2016
 * Last modified: Mon Dec 06 12:59:10 2021
 * Model Version: 0.3.0
 * Description: Thermal reactor start time reduction function

   Outstandings:
   -------------
   - NA
 * modified Comment: V0.1.0 18.05.2021 Maran   TrStRed function first draft
   V0.1.1 27.05.2021 Maran   added limitation based on cyl. EG max temp. above setpoint
   V0.1.2 02.08.2021 Maran   added half load factor for function limit range
   V0.2.0 15.11.2021 Maran   added saturation limits to control error for the closed loop integrator (PERM parameters)
   V0.3.0 06.12.2021 Maran   removed unused logic in controller block; added filtered value of monitoring variables in debug interface
 ********************************************************************
 * Implementation of program TrStRed
 ********************************************************************
 * Generated with B&R Automation Studio Target for Simulink V6.3.1
 * (ERT based)
 ********************************************************************/

#include <bur/plctypes.h>
#include "TrStRed.h"
#include "rtwtypes.h"

/* Defines */
#define SS_TERMINATE 4
#define SS_OUTPUT 3
#define SS_INITIALIZE 2

/*  Data Types */

/**************************** GLOBAL DATA *************************************/
/*  Definitions */

/*  Declarations  */

/***************************** FILE SCOPE DATA ********************************/

/*************************** FUNCTIONS ****************************************/
#ifdef __cplusplus

unsigned long bur_heap_size = 6553500;

#endif

/*LEGACYMODE_VARIABLES*/
void fTrStRed(struct fTrStRed* inst)
{
  tag_RTM_TrStRed* const TrStRed_M = &(inst)->bur_TrStRed;
	inst->bur_TrStRed.blockIO = &(inst)->bur_BlockIO_TrStRed;
	inst->bur_TrStRed.prevZCSigState = &(inst)->bur_PrevZCSigStates_TrStRed;
	inst->bur_TrStRed.inputs = &(inst)->bur_ExternalInputs_TrStRed;
	inst->bur_TrStRed.outputs = &(inst)->bur_ExternalOutputs_TrStRed;
	inst->bur_TrStRed.dwork = &(inst)->bur_D_Work_TrStRed;

  switch (inst->ssMethodType)
  {
   case SS_INITIALIZE:
    /* call model initialize function */
    TrStRed_initialize(TrStRed_M, inst);
    break;

   case SS_OUTPUT:
    /* call model step function */
    TrStRed_step(TrStRed_M, inst);

    break;

   case SS_TERMINATE:
    /* call model terminate function */
    TrStRed_terminate(TrStRed_M, inst);
    break;
  }
}

/*****************************************************************************
   Function block sample time: 0.01s
 *****************************************************************************/

/*****************************************************************************
   B&R Automation Studio Target for Simulink Version: A6.3.1 (15-Dec-2020)
 *****************************************************************************/

/*======================== TOOL VERSION INFORMATION ==========================*
 * MATLAB 9.8 (R2020a)18-Nov-2019                                             *
 * Simulink 10.1 (R2020a)18-Nov-2019                                          *
 * Simulink Coder 9.3 (R2020a)18-Nov-2019                                     *
 * Embedded Coder 7.4 (R2020a)18-Nov-2019                                     *
 * Stateflow 10.2 (R2020a)18-Nov-2019                                         *
 *============================================================================*/

/*======================= LICENSE IN USE INFORMATION =========================*
 * matlab                                                                     *
 * matlab_coder                                                               *
 * real-time_workshop                                                         *
 * rtw_embedded_coder                                                         *
 * simulink                                                                   *
 *============================================================================*/
```

#### lTrStRed.fun
```iecst
FUNCTION_BLOCK fTrStRed
  VAR_INPUT
    ssMethodType: SINT;
  END_VAR
  VAR_INPUT
        Perm : TrStRed_PERM_Bus; (**)
  END_VAR
  VAR_INPUT
        In : TrStRed_IN_Bus; (**)
  END_VAR
  VAR_INPUT
        Para : TrStRed_PARA_Bus; (**)
  END_VAR
  VAR_OUTPUT
        Out : TrStRed_OUT_Bus; (**)
  END_VAR
  VAR_OUTPUT
        Dbg : TrStRed_DBG_Bus; (**)
  END_VAR
  VAR_OUTPUT
        Version : UDINT := 0; (**)
  END_VAR
	VAR
		bur_BlockIO_TrStRed : BlockIO_TrStRed;
	END_VAR
	VAR
		bur_PrevZCSigStates_TrStRed : PrevZCSigStates_TrStRed;
	END_VAR
	VAR
		bur_ExternalInputs_TrStRed : ExternalInputs_TrStRed;
	END_VAR
	VAR
		bur_ExternalOutputs_TrStRed : ExternalOutputs_TrStRed;
	END_VAR
	VAR
		bur_D_Work_TrStRed : D_Work_TrStRed;
	END_VAR
	VAR
		bur_TrStRed : tag_RTM_TrStRed;
	END_VAR
END_FUNCTION_BLOCK
```

#### lTrStRed.typ
```iecst
TYPE
	TrStRed_DBG_Bus :  STRUCT
		rT_CtrlError :  REAL; (*Error between target and actual EG max temperature (degC)*)
		rCA_IP_Lim_preSat :  REAL; (*relative ITP upper limit before saturation (degCA)*)
		bInternalLimitAct :  BOOL; (*true, if TrStRed internal saturation limitation active ()*)
		rCtrl_Int_InputPreGain :  REAL; (*control integrator input before integral gain (degC)*)
		rPr_Leanox_Dev_filt :  REAL; (*filtered Leanox controller deviation (mbar)*)
		rIgnVolt_Max_filt :  REAL; (*filtered maximum ignition voltage (kV)*)
		rCtrl_IntegrInput :  REAL; (*actual control integrator input (degCA/s)*)
		bSteadyState :  BOOL; (*true, if engine power steady as per TrStRed definition ()*)
		rCA_LowLimit_Act :  REAL; (*actual control limit TrStRed function - relative ITP (degCA)*)
	END_STRUCT;

	TrStRed_IN_Bus :  STRUCT
		bTrStRed_active :  BOOL; (*TrStRed function activation conditions ()*)
		rP_Norm :  REAL; (*normalized and filtered actual power (%)*)
		rP_Set_Norm :  REAL; (*normalized power setpoint (%)*)
		rPr_Leanox_Dev :  REAL; (*Leanox controller deviation (mbar)*)
		rT_EG_CylMax :  REAL; (*cylinder temperature maximal value (degC)*)
		rT_EG_MaxLimit :  REAL; (*exhaust gas temperature maximum limit (degC)*)
		rT_EG_CylAvg :  REAL; (*cylinder temperature average (degC)*)
		rMisfire_level :  REAL; (*misfire integrator value (%)*)
		rIgnVolt_Max :  REAL; (*maximum ignition voltage (kV)*)
		rCA_Ign_UpLim :  REAL; (*highest relative ITP of all cylinders (degCA)*)
		rCA_IgnP_relAw :  REAL; (*relative ITP feedback (degCA)*)
		rT_EGbTC :  REAL; (*exhaust gas temperature before turbo charger T3 (degC)*)
		bThR_RelGas :  BOOL; (*Thermal Reactor auxiliary gas injection ()*)
		bReset :  BOOL; (*Reset TrStRed function ()*)
		bCycleReset :  BOOL; (*Reset TrStRed operating cycle ()*)
	END_STRUCT;

	TrStRed_OUT_Bus :  STRUCT
		rCA_IP_Lim :  REAL; (*relative ITP upper limit (degCA)*)
		bCycleStarted :  BOOL; (*TrStRed operating cycle started ()*)
		bCycleCompleted :  BOOL; (*TrStRed operating cycle completed ()*)
		bTrStRed_Stop :  BOOL; (*TrStRed function stop mode ()*)
	END_STRUCT;

	TrStRed_PARA_Bus :  STRUCT
		rT_EG_Avg_HiLim :  REAL; (*cylinder temperature average high limit (degC)*)
		rT_EG_Max_LimMarg :  REAL; (*margin from max. cyl. temperature for controller setpoint (degC)*)
		rIgnVoltMax_Lim :  REAL; (*maximum ignition voltage (kV)*)
		rT_EGbTC_HiLim :  REAL; (*turbocharger inlet temperature high warning (degC)*)
		rCA_TrStRed_LowLimit :  REAL; (*control limit TrStRed function - relative ITP (degCA)*)
		rGain_TrStRed_halfLoadLim :  REAL; (*half load factor for TrStRed function control limit (%)*)
	END_STRUCT;

	TrStRed_PERM_Bus :  STRUCT
		rCA_RateLimit :  REAL; (*TrStRed function output rate limiter (degCA/s)*)
		rMisfire_Lim :  REAL; (*misfire threshold - function internal limitations (%)*)
		rPr_LxDev_Lim :  REAL; (*Leanox deviation max. threshold - function internal limitations (mbar)*)
		rFiltConst_LxDev :  REAL; (*filter coefficient PT1 - Leanox deviation - function internal limitations (s)*)
		rFiltConst_IgnVolt :  REAL; (*filter coefficient PT1 - ignition voltage - function internal limitations (s)*)
		rIgnVolt_LimMarg :  REAL; (*ignition voltage max exceedance from warning limit - function internal limitations (kV)*)
		rT_EG_Avg_LimMarg :  REAL; (*cylinder temperature average margin from high limit - function internal limitations (degC)*)
		rT_EGbTC_LimMarg :  REAL; (*turbocharger inlet temperature margin from high warning - function internal limitations (degC)*)
		iTimerDelay_Steady :  UINT; (*delay timer for TrStRed steady state (s)*)
		rP_diffThres_Steady :  REAL; (*normalized power setpoint/actual difference for TrStRed steady state (%)*)
		rCtrl_ki :  REAL; (*ctrl integral gain (degCA/degC/s)*)
		iStopTimer :  UINT; (*time delay for TrStRed function stop at reactor temperature target (s)*)
		rCtrl_kAw :  REAL; (*ctrl antiwind-up gain for integrator (degC/degCA)*)
		rLimitsReleaseFactor :  REAL; (*factor for releasing internal protection limitations referred to main rate limiter ()*)
		rT_EG_Max_LimOffset :  REAL; (*offset to max. cyl. temperature referred to limit value - function internal limitations (degC)*)
		rT_CtrlError_UpLim :  REAL; (*Upper saturation limit for control error (degC)*)
		rT_CtrlError_LowLim :  REAL; (*Lower saturation limit for control error (degC)*)
	END_STRUCT;

END_TYPE

TYPE
rtB_Filter_TrStRed : STRUCT
	Switch : REAL;
END_STRUCT;
rtDW_Filter_TrStRed : STRUCT
	DiscreteTimeIntegrator_DSTATE : REAL;
	DiscreteTimeIntegrator_PrevRese : SINT;
	DiscreteTimeIntegrator_IC_LOADI : USINT;
END_STRUCT;
rtB_TON_TrStRed : STRUCT
	LogicalOperator3 : BOOL;
END_STRUCT;
rtDW_TON_TrStRed : STRUCT
	DiscreteTimeIntegrator_DSTATE : UINT;
	DiscreteTimeIntegrator_PrevRese : SINT;
END_STRUCT;
BlockIO_TrStRed : STRUCT
	BusInput1 : TrStRed_PERM_Bus;
	BusInput2 : TrStRed_IN_Bus;
	BusInput : TrStRed_PARA_Bus;
	UnitDelay : UDINT;
	TON_k : rtB_TON_TrStRed;
	TON : rtB_TON_TrStRed;
	Filter1 : rtB_Filter_TrStRed;
	Filter : rtB_Filter_TrStRed;
END_STRUCT;
D_Work_TrStRed : STRUCT
	ITCtrUi : REAL;
	Delay_DSTATE : REAL;
	Delay_DSTATE_b : REAL;
	UnitDelay1_DSTATE : REAL;
	UnitDelay_DSTATE : UDINT;
	UnitDelay_DSTATE_j : BOOL;
	DiscreteTimeIntegrator_PrevRese : SINT;
	DiscreteTimeIntegrator_IC_LOADI : USINT;
	icLoad : USINT;
	icLoad_l : USINT;
	Memory_PreviousInput : BOOL;
	Memory_PreviousInput_o : BOOL;
	Memory_PreviousInput_l : BOOL;
	TON_k : rtDW_TON_TrStRed;
	TON : rtDW_TON_TrStRed;
	Filter1 : rtDW_Filter_TrStRed;
	Filter : rtDW_Filter_TrStRed;
END_STRUCT;
PrevZCSigStates_TrStRed : STRUCT
	Delay_Reset_ZCE : USINT;
	Delay_Reset_ZCE_l : USINT;
END_STRUCT;
rtC_Filter_TrStRed : STRUCT
	Conversion : REAL;
END_STRUCT;
ConstBlockIO_TrStRed : STRUCT
	Filter1 : rtC_Filter_TrStRed;
	Filter : rtC_Filter_TrStRed;
END_STRUCT;
ConstParam_TrStRed : STRUCT
	pooled10 : ARRAY[0..15] OF BOOL;
END_STRUCT;
ExternalInputs_TrStRed : STRUCT
	In : TrStRed_IN_Bus;
	Para : TrStRed_PARA_Bus;
	Perm : TrStRed_PERM_Bus;
END_STRUCT;
ExternalOutputs_TrStRed : STRUCT
	Out : TrStRed_OUT_Bus;
	dbg : TrStRed_DBG_Bus;
END_STRUCT;
tag_RTM_TrStRed : STRUCT
	errorStatus : REFERENCE TO USINT;
	blockIO : REFERENCE TO BlockIO_TrStRed;
	prevZCSigState : REFERENCE TO PrevZCSigStates_TrStRed;
	inputs : REFERENCE TO ExternalInputs_TrStRed;
	outputs : REFERENCE TO ExternalOutputs_TrStRed;
	dwork : REFERENCE TO D_Work_TrStRed;
END_STRUCT;
RT_MODEL_TrStRed : tag_RTM_TrStRed;

END_TYPE
TYPE
END_TYPE
```

#### lib_properties.txt
```
For manual assignment to hardware configuration please
add the following additional include directories:

\Logical\MATLAB_includes\R2020a\

And the following additional build options:

-lm -D MODEL=TrStRed -D NUMST=1 -D NCSTATES=0 -D HAVESTDIO -D MODEL_HAS_DYNAMICALLY_LOADED_SFCNS=0 -D CLASSIC_INTERFACE=0 -D ALLOCATIONFCN=0 -D TID01EQ=0 -D TERMFCN=1 -D ONESTEPFCN=1 -D MAT_FILE=0 -D MULTI_INSTANCE_CODE=1 -D INTEGER_CODE=0 -D MT=0
```

#### rt_defines.h
```c
/********************************************************************
 * COPYRIGHT -- B&R Industrial Automation GmbH
 ********************************************************************
 * Program: TrStRed
 * File: rt_defines.h
 * Author: 105055527
 * Last modified by: maranen00
 * Created: Mon Sep 05 18:14:57 2016
 * Last modified: Mon Dec 06 12:59:10 2021
 * Model Version: 0.3.0
 * Description: Thermal reactor start time reduction function

   Outstandings:
   -------------
   - NA
 * modified Comment: V0.1.0 18.05.2021 Maran   TrStRed function first draft
   V0.1.1 27.05.2021 Maran   added limitation based on cyl. EG max temp. above setpoint
   V0.1.2 02.08.2021 Maran   added half load factor for function limit range
   V0.2.0 15.11.2021 Maran   added saturation limits to control error for the closed loop integrator (PERM parameters)
   V0.3.0 06.12.2021 Maran   removed unused logic in controller block; added filtered value of monitoring variables in debug interface
 ********************************************************************
 * Header for program TrStRed
 ********************************************************************
 * Generated with B&R Automation Studio Target for Simulink V6.3.1
 * (ERT based)
 ********************************************************************/

#ifndef RTW_HEADER_rt_defines_h_
#define RTW_HEADER_rt_defines_h_
#ifndef MIN
#define MIN(a,b)                       ((a) < (b) ? (a) : (b))
#endif

#ifndef MAX
#define MAX(a,b)                       ((a) > (b) ? (a) : (b))
#endif

#ifndef AST_ROUND
#define AST_ROUND(x)                   ((x)>=0?(long long)((x)+0.5):(long long)((x)-0.5))
#endif

/*===========*
 * Constants *
 *===========*/
#define RT_PI                          3.14159265358979323846
#define RT_PIF                         3.1415927F
#define RT_LN_10                       2.30258509299404568402
#define RT_LN_10F                      2.3025851F
#define RT_LOG10E                      0.43429448190325182765
#define RT_LOG10EF                     0.43429449F
#define RT_E                           2.7182818284590452354
#define RT_EF                          2.7182817F

/*
 * UNUSED_PARAMETER(x)
 *   Used to specify that a function parameter (argument) is required but not
 *   accessed by the function body.
 */
#ifndef UNUSED_PARAMETER
# if defined(__LCC__)
#   define UNUSED_PARAMETER(x)                                   /* do nothing */
# else

/*
 * This is the semi-ANSI standard way of indicating that an
 * unused function parameter is required.
 */
#   define UNUSED_PARAMETER(x)         (void) (x)
# endif
#endif
#endif                                 /* RTW_HEADER_rt_defines_h_ */
```
